LIN {X 0,Y 360.383,Z 396.223,A -85,B 0,C 180,E1 -13044.404,E2 -13044.404} C_VEL
LIN {X 0,Y 360.363,Z 398.205,A -85,B 0,C 180,E1 -13045.526,E2 -13045.526} C_VEL
LIN {X 0,Y 360.299,Z 399.765,A -85,B 0,C 180,E1 -13046.645,E2 -13046.645} C_VEL
LIN {X 0,Y 360.265,Z 400.875,A -85,B 0,C 180,E1 -13047.764,E2 -13047.764} C_VEL
LIN {X 0,Y 360.317,Z 401.567,A -85,B 0,C 180,E1 -13048.882,E2 -13048.882} C_VEL
LIN {X 0,Y 360.36,Z 401.867,A -85,B 0,C 180,E1 -13050,E2 -13050} C_VEL
LIN {X 0,Y 360.303,Z 401.773,A -85,B 0,C 180,E1 -13051.118,E2 -13051.118} C_VEL
LIN {X 0,Y 360.263,Z 401.25,A -85,B 0,C 180,E1 -13052.236,E2 -13052.236} C_VEL
LIN {X 0,Y 360.296,Z 400.314,A -85,B 0,C 180,E1 -13053.355,E2 -13053.355} C_VEL
LIN {X 0,Y 360.346,Z 398.979,A -85,B 0,C 180,E1 -13054.474,E2 -13054.474} C_VEL
LIN {X 0,Y 360.378,Z 396.542,A -85,B 0,C 180,E1 -13055.961,E2 -13055.961} C_VEL
LIN {X 0,Y 360.672,Z 392.315,A -85,B 0,C 180,E1 -13057.84,E2 -13057.84} C_VEL
LIN {X 0,Y 361.093,Z 387.341,A -85,B 0,C 180,E1 -13059.523,E2 -13059.523} C_VEL
LIN {X 0,Y 361.704,Z 381.091,A -85,B 0,C 180,E1 -13061.204,E2 -13061.204} C_VEL
LIN {X 0,Y 362.687,Z 373.329,A -85,B 0,C 180,E1 -13062.876,E2 -13062.876} C_VEL
LIN {X 0,Y 363.599,Z 365.4,A -85,B 0,C 180,E1 -13064.267,E2 -13064.267} C_VEL
LIN {X 0,Y 364.63,Z 355.745,A -85,B 0,C 180,E1 -13065.655,E2 -13065.655} C_VEL
LIN {X 0,Y 365.809,Z 345.051,A -85,B 0,C 180,E1 -13066.893,E2 -13066.893} C_VEL
LIN {X 0,Y 366.862,Z 334.733,A -85,B 0,C 180,E1 -13067.849,E2 -13067.849} C_VEL
LIN {X 0,Y 367.953,Z 323.553,A -85,B 0,C 180,E1 -13068.659,E2 -13068.659} C_VEL
LIN {X 0,Y 368.836,Z 310.34,A -85,B 0,C 180,E1 -13069.37,E2 -13069.37} C_VEL
LIN {X 0,Y 369.589,Z 297.288,A -85,B 0,C 180,E1 -13069.835,E2 -13069.835} C_VEL
LIN {X 0,Y 370.935,Z 222.024,A -85,B 0,C 180,E1 -13071.405,E2 -13071.405} C_VEL
LIN {X 0,Y 367.136,Z 199.174,A -85,B 0,C 180,E1 -13072.171,E2 -13072.171} C_VEL
LIN {X 0,Y 365.04,Z 188.802,A -85,B 0,C 180,E1 -13072.56,E2 -13072.56} C_VEL
LIN {X 0,Y 366.009,Z 179.574,A -85,B 0,C 180,E1 -13074.686,E2 -13074.686} C_VEL
LIN {X 0,Y 365.116,Z 173.255,A -85,B 0,C 180,E1 -13076.278,E2 -13076.278} C_VEL
LIN {X 0,Y 362.68,Z 161.895,A -85,B 0,C 180,E1 -13079.307,E2 -13079.307} C_VEL
LIN {X 0,Y 361.904,Z 158.409,A -85,B 0,C 180,E1 -13080.325,E2 -13080.325} C_VEL
LIN {X 0,Y 361.851,Z 158.414,A -85,B 0,C 180,E1 -13084.281,E2 -13084.281} C_VEL
LIN {X 0,Y 361.857,Z 158.413,A -85,B 0,C 180,E1 -13087.221,E2 -13087.221} C_VEL
LIN {X 0,Y 361.812,Z 158.419,A -85,B 0,C 180,E1 -13090.751,E2 -13090.751} C_VEL
LIN {X 0,Y 361.813,Z 158.416,A -85,B 0,C 180,E1 -13094.37,E2 -13094.37} C_VEL
LIN {X 0,Y 361.824,Z 158.414,A -85,B 0,C 180,E1 -13097.571,E2 -13097.571} C_VEL
LIN {X 0,Y 361.842,Z 158.412,A -85,B 0,C 180,E1 -13101.572,E2 -13101.572} C_VEL
LIN {X 0,Y 361.872,Z 158.408,A -85,B 0,C 180,E1 -13104.657,E2 -13104.657} C_VEL
LIN {X 0,Y 361.839,Z 158.41,A -85,B 0,C 180,E1 -13108.371,E2 -13108.371} C_VEL
LIN {X 0,Y 361.851,Z 158.404,A -85,B 0,C 180,E1 -13110.951,E2 -13110.951} C_VEL
LIN {X 0,Y 361.853,Z 158.403,A -85,B 0,C 180,E1 -13114.704,E2 -13114.704} C_VEL
LIN {X 0,Y 361.855,Z 158.408,A -85,B 0,C 180,E1 -13118.345,E2 -13118.345} C_VEL
LIN {X 0,Y 361.907,Z 158.405,A -85,B 0,C 180,E1 -13122.093,E2 -13122.093} C_VEL
LIN {X 0,Y 361.967,Z 158.398,A -85,B 0,C 180,E1 -13126.527,E2 -13126.527} C_VEL
LIN {X 0,Y 361.996,Z 158.385,A -85,B 0,C 180,E1 -13129.937,E2 -13129.937} C_VEL
LIN {X 0,Y 362.094,Z 158.377,A -85,B 0,C 180,E1 -13132.191,E2 -13132.191} C_VEL
LIN {X 0,Y 362.09,Z 158.375,A -85,B 0,C 180,E1 -13134.431,E2 -13134.431} C_VEL
LIN {X 0,Y 362.261,Z 158.351,A -85,B 0,C 180,E1 -13137.776,E2 -13137.776} C_VEL
LIN {X 0,Y 362.177,Z 158.365,A -85,B 0,C 180,E1 -13141.112,E2 -13141.112} C_VEL
LIN {X 0,Y 362.261,Z 158.354,A -85,B 0,C 180,E1 -13142.224,E2 -13142.224} C_VEL
LIN {X 0,Y 362.122,Z 158.376,A -85,B 0,C 180,E1 -13146.687,E2 -13146.687} C_VEL
LIN {X 0,Y 361.999,Z 158.391,A -85,B 0,C 180,E1 -13150.063,E2 -13150.063} C_VEL
LIN {X 0,Y 361.983,Z 158.397,A -85,B 0,C 180,E1 -13153.887,E2 -13153.887} C_VEL
LIN {X 0,Y 361.887,Z 158.405,A -85,B 0,C 180,E1 -13158.103,E2 -13158.103} C_VEL
LIN {X 0,Y 361.857,Z 158.414,A -85,B 0,C 180,E1 -13161.655,E2 -13161.655} C_VEL
LIN {X 0,Y 361.864,Z 158.414,A -85,B 0,C 180,E1 -13165.295,E2 -13165.295} C_VEL
LIN {X 0,Y 361.858,Z 158.412,A -85,B 0,C 180,E1 -13169.074,E2 -13169.074} C_VEL
LIN {X 0,Y 361.91,Z 158.531,A -85,B 0,C 180,E1 -13171.786,E2 -13171.786} C_VEL
LIN {X 0,Y 364.366,Z 169.922,A -85,B 0,C 180,E1 -13175.018,E2 -13175.018} C_VEL
LIN {X 0,Y 364.756,Z 171.823,A -85,B 0,C 180,E1 -13175.482,E2 -13175.482} C_VEL
LIN {X 0,Y 367.896,Z 180.526,A -85,B 0,C 180,E1 -13175.908,E2 -13175.908} C_VEL
LIN {X 0,Y 371.495,Z 197.463,A -85,B 0,C 180,E1 -13176.537,E2 -13176.537} C_VEL
LIN {X 0,Y 369.759,Z 279.168,A -85,B 0,C 180,E1 -13178.23,E2 -13178.23} C_VEL
LIN {X 0,Y 369.129,Z 292.46,A -85,B 0,C 180,E1 -13178.721,E2 -13178.721} C_VEL
LIN {X 0,Y 368.436,Z 305.031,A -85,B 0,C 180,E1 -13179.416,E2 -13179.416} C_VEL
LIN {X 0,Y 367.469,Z 316.572,A -85,B 0,C 180,E1 -13180.272,E2 -13180.272} C_VEL
LIN {X 0,Y 366.343,Z 328.059,A -85,B 0,C 180,E1 -13181.373,E2 -13181.373} C_VEL
LIN {X 0,Y 365.194,Z 338.479,A -85,B 0,C 180,E1 -13182.626,E2 -13182.626} C_VEL
LIN {X 0,Y 364.038,Z 348.321,A -85,B 0,C 180,E1 -13184.112,E2 -13184.112} C_VEL
LIN {X 0,Y 362.998,Z 357.318,A -85,B 0,C 180,E1 -13185.813,E2 -13185.813} C_VEL
LIN {X 0,Y 362.078,Z 364.557,A -85,B 0,C 180,E1 -13187.527,E2 -13187.527} C_VEL
LIN {X 0,Y 361.392,Z 370.511,A -85,B 0,C 180,E1 -13189.327,E2 -13189.327} C_VEL
LIN {X 0,Y 360.886,Z 375.198,A -85,B 0,C 180,E1 -13191.167,E2 -13191.167} C_VEL
LIN {X 0,Y 360.496,Z 378.709,A -85,B 0,C 180,E1 -13193.065,E2 -13193.065} C_VEL
LIN {X 0,Y 360.179,Z 381.055,A -85,B 0,C 180,E1 -13195.038,E2 -13195.038} C_VEL
LIN {X 0,Y 360.074,Z 382.107,A -85,B 0,C 180,E1 -13197.065,E2 -13197.065} C_VEL
LIN {X 0,Y 360.104,Z 381.816,A -85,B 0,C 180,E1 -13199.175,E2 -13199.175} C_VEL
LIN {X 0,Y 360.268,Z 380.007,A -85,B 0,C 180,E1 -13201.384,E2 -13201.384} C_VEL
LIN {X 0,Y 360.569,Z 376.96,A -85,B 0,C 180,E1 -13203.365,E2 -13203.365} C_VEL
LIN {X 0,Y 360.916,Z 372.764,A -85,B 0,C 180,E1 -13205.25,E2 -13205.25} C_VEL
LIN {X 0,Y 361.336,Z 367.249,A -85,B 0,C 180,E1 -13207.107,E2 -13207.107} C_VEL
LIN {X 0,Y 361.938,Z 360.996,A -85,B 0,C 180,E1 -13208.757,E2 -13208.757} C_VEL
LIN {X 0,Y 362.777,Z 352.79,A -85,B 0,C 180,E1 -13210.477,E2 -13210.477} C_VEL
LIN {X 0,Y 363.701,Z 343.833,A -85,B 0,C 180,E1 -13211.99,E2 -13211.99} C_VEL
LIN {X 0,Y 364.645,Z 334.126,A -85,B 0,C 180,E1 -13213.321,E2 -13213.321} C_VEL
LIN {X 0,Y 365.693,Z 322.992,A -85,B 0,C 180,E1 -13214.535,E2 -13214.535} C_VEL
LIN {X 0,Y 366.566,Z 311.016,A -85,B 0,C 180,E1 -13215.567,E2 -13215.567} C_VEL
LIN {X 0,Y 367.308,Z 298.616,A -85,B 0,C 180,E1 -13216.374,E2 -13216.374} C_VEL
LIN {X 0,Y 368.004,Z 285.25,A -85,B 0,C 180,E1 -13216.981,E2 -13216.981} C_VEL
LIN {X 0,Y 368.435,Z 272.362,A -85,B 0,C 180,E1 -13217.347,E2 -13217.347} C_VEL
LIN {X 0,Y 369.683,Z 196.406,A -85,B 0,C 180,E1 -13218.884,E2 -13218.884} C_VEL
LIN {X 0,Y 364.942,Z 172.85,A -85,B 0,C 180,E1 -13219.651,E2 -13219.651} C_VEL
LIN {X 0,Y 364.418,Z 171.078,A -85,B 0,C 180,E1 -13219.724,E2 -13219.724} C_VEL
LIN {X 0,Y 362.13,Z 158.379,A -85,B 0,C 180,E1 -13223.243,E2 -13223.243} C_VEL
LIN {X 0,Y 362.279,Z 158.355,A -85,B 0,C 180,E1 -13227.776,E2 -13227.776} C_VEL
LIN {X 0,Y 362.206,Z 158.364,A -85,B 0,C 180,E1 -13231.112,E2 -13231.112} C_VEL
LIN {X 0,Y 362.267,Z 158.361,A -85,B 0,C 180,E1 -13232.224,E2 -13232.224} C_VEL
LIN {X 0,Y 362.124,Z 158.376,A -85,B 0,C 180,E1 -13236.687,E2 -13236.687} C_VEL
LIN {X 0,Y 362.03,Z 158.391,A -85,B 0,C 180,E1 -13240.062,E2 -13240.062} C_VEL
LIN {X 0,Y 361.973,Z 158.392,A -85,B 0,C 180,E1 -13240.987,E2 -13240.987} C_VEL
LIN {X 0,Y 361.296,Z 158.481,A -85,B 0,C 180,E1 -13241.916,E2 -13241.916} C_VEL
LIN {X 0,Y 358.408,Z 158.838,A -85,B 0,C 180,E1 -13243.426,E2 -13243.426} C_VEL
LIN {X 0,Y 355.968,Z 159.142,A -85,B 0,C 180,E1 -13244.648,E2 -13244.648} C_VEL
LIN {X 0,Y 354.927,Z 159.273,A -85,B 0,C 180,E1 -13245.594,E2 -13245.594} C_VEL
LIN {X 0,Y 354.847,Z 159.283,A -85,B 0,C 180,E1 -13245.914,E2 -13245.914} C_VEL
LIN {X 0,Y 354.849,Z 159.281,A -85,B 0,C 180,E1 -13248.475,E2 -13248.475} C_VEL
LIN {X 0,Y 354.809,Z 159.288,A -85,B 0,C 180,E1 -13252.108,E2 -13252.108} C_VEL
LIN {X 0,Y 354.805,Z 159.291,A -85,B 0,C 180,E1 -13255.835,E2 -13255.835} C_VEL
LIN {X 0,Y 354.798,Z 159.292,A -85,B 0,C 180,E1 -13259.684,E2 -13259.684} C_VEL
LIN {X 0,Y 354.789,Z 159.288,A -85,B 0,C 180,E1 -13262.334,E2 -13262.334} C_VEL
LIN {X 0,Y 354.823,Z 159.287,A -85,B 0,C 180,E1 -13265.699,E2 -13265.699} C_VEL
LIN {X 0,Y 354.77,Z 159.296,A -85,B 0,C 180,E1 -13269.413,E2 -13269.413} C_VEL
LIN {X 0,Y 354.787,Z 159.29,A -85,B 0,C 180,E1 -13272.867,E2 -13272.867} C_VEL
LIN {X 0,Y 354.765,Z 159.291,A -85,B 0,C 180,E1 -13276.103,E2 -13276.103} C_VEL
LIN {X 0,Y 354.768,Z 159.296,A -85,B 0,C 180,E1 -13279.176,E2 -13279.176} C_VEL
LIN {X 0,Y 354.802,Z 159.286,A -85,B 0,C 180,E1 -13282.404,E2 -13282.404} C_VEL
LIN {X 0,Y 354.811,Z 159.29,A -85,B 0,C 180,E1 -13284.94,E2 -13284.94} C_VEL
LIN {X 0,Y 354.796,Z 159.288,A -85,B 0,C 180,E1 -13288.405,E2 -13288.405} C_VEL
LIN {X 0,Y 354.802,Z 159.286,A -85,B 0,C 180,E1 -13291.615,E2 -13291.615} C_VEL
LIN {X 0,Y 354.837,Z 159.282,A -85,B 0,C 180,E1 -13295.657,E2 -13295.657} C_VEL
LIN {X 0,Y 354.827,Z 159.285,A -85,B 0,C 180,E1 -13299.113,E2 -13299.113} C_VEL
LIN {X 0,Y 354.855,Z 159.284,A -85,B 0,C 180,E1 -13302.718,E2 -13302.718} C_VEL
LIN {X 0,Y 354.943,Z 159.272,A -85,B 0,C 180,E1 -13306.255,E2 -13306.255} C_VEL
LIN {X 0,Y 354.958,Z 159.267,A -85,B 0,C 180,E1 -13309.735,E2 -13309.735} C_VEL
LIN {X 0,Y 355.091,Z 159.25,A -85,B 0,C 180,E1 -13313.18,E2 -13313.18} C_VEL
LIN {X 0,Y 355.23,Z 159.234,A -85,B 0,C 180,E1 -13317.732,E2 -13317.732} C_VEL
LIN {X 0,Y 355.149,Z 159.243,A -85,B 0,C 180,E1 -13321.134,E2 -13321.134} C_VEL
LIN {X 0,Y 355.229,Z 159.238,A -85,B 0,C 180,E1 -13322.268,E2 -13322.268} C_VEL
LIN {X 0,Y 355.091,Z 159.25,A -85,B 0,C 180,E1 -13326.82,E2 -13326.82} C_VEL
LIN {X 0,Y 354.953,Z 159.27,A -85,B 0,C 180,E1 -13330.265,E2 -13330.265} C_VEL
LIN {X 0,Y 354.895,Z 159.279,A -85,B 0,C 180,E1 -13333.986,E2 -13333.986} C_VEL
LIN {X 0,Y 354.837,Z 159.285,A -85,B 0,C 180,E1 -13338.064,E2 -13338.064} C_VEL
LIN {X 0,Y 354.808,Z 159.287,A -85,B 0,C 180,E1 -13342.108,E2 -13342.108} C_VEL
LIN {X 0,Y 354.797,Z 159.29,A -85,B 0,C 180,E1 -13345.835,E2 -13345.835} C_VEL
LIN {X 0,Y 354.795,Z 159.291,A -85,B 0,C 180,E1 -13349.684,E2 -13349.684} C_VEL
LIN {X 0,Y 354.788,Z 159.288,A -85,B 0,C 180,E1 -13352.333,E2 -13352.333} C_VEL
LIN {X 0,Y 354.82,Z 159.286,A -85,B 0,C 180,E1 -13355.698,E2 -13355.698} C_VEL
LIN {X 0,Y 354.77,Z 159.294,A -85,B 0,C 180,E1 -13359.412,E2 -13359.412} C_VEL
LIN {X 0,Y 354.783,Z 159.292,A -85,B 0,C 180,E1 -13362.866,E2 -13362.866} C_VEL
LIN {X 0,Y 354.764,Z 159.291,A -85,B 0,C 180,E1 -13366.103,E2 -13366.103} C_VEL
LIN {X 0,Y 354.764,Z 159.295,A -85,B 0,C 180,E1 -13369.175,E2 -13369.175} C_VEL
LIN {X 0,Y 354.8,Z 159.288,A -85,B 0,C 180,E1 -13372.404,E2 -13372.404} C_VEL
LIN {X 0,Y 354.809,Z 159.29,A -85,B 0,C 180,E1 -13374.94,E2 -13374.94} C_VEL
LIN {X 0,Y 354.777,Z 159.292,A -85,B 0,C 180,E1 -13378.41,E2 -13378.41} C_VEL
LIN {X 0,Y 354.854,Z 159.395,A -85,B 0,C 180,E1 -13380.321,E2 -13380.321} C_VEL
LIN {X 0,Y 357.448,Z 172.358,A -85,B 0,C 180,E1 -13383.744,E2 -13383.744} C_VEL
LIN {X 0,Y 358.451,Z 178.801,A -85,B 0,C 180,E1 -13385.377,E2 -13385.377} C_VEL
LIN {X 0,Y 357.438,Z 189.546,A -85,B 0,C 180,E1 -13387.906,E2 -13387.906} C_VEL
LIN {X 0,Y 362.684,Z 223.59,A -85,B 0,C 180,E1 -13388.946,E2 -13388.946} C_VEL
LIN {X 0,Y 361.286,Z 298.073,A -85,B 0,C 180,E1 -13390.504,E2 -13390.504} C_VEL
LIN {X 0,Y 360.646,Z 311.829,A -85,B 0,C 180,E1 -13391.023,E2 -13391.023} C_VEL
LIN {X 0,Y 359.793,Z 324.254,A -85,B 0,C 180,E1 -13391.714,E2 -13391.714} C_VEL
LIN {X 0,Y 358.739,Z 336.164,A -85,B 0,C 180,E1 -13392.617,E2 -13392.617} C_VEL
LIN {X 0,Y 357.646,Z 347.626,A -85,B 0,C 180,E1 -13393.738,E2 -13393.738} C_VEL
LIN {X 0,Y 356.733,Z 357.74,A -85,B 0,C 180,E1 -13394.981,E2 -13394.981} C_VEL
LIN {X 0,Y 355.837,Z 366.43,A -85,B 0,C 180,E1 -13396.29,E2 -13396.29} C_VEL
LIN {X 0,Y 354.87,Z 375.592,A -85,B 0,C 180,E1 -13397.998,E2 -13397.998} C_VEL
LIN {X 0,Y 354.199,Z 382.972,A -85,B 0,C 180,E1 -13399.713,E2 -13399.713} C_VEL
LIN {X 0,Y 353.712,Z 388.878,A -85,B 0,C 180,E1 -13401.43,E2 -13401.43} C_VEL
LIN {X 0,Y 353.415,Z 393.517,A -85,B 0,C 180,E1 -13403.147,E2 -13403.147} C_VEL
LIN {X 0,Y 353.29,Z 395.958,A -85,B 0,C 180,E1 -13404.292,E2 -13404.292} C_VEL
LIN {X 0,Y 353.276,Z 397.953,A -85,B 0,C 180,E1 -13405.436,E2 -13405.436} C_VEL
LIN {X 0,Y 353.221,Z 399.525,A -85,B 0,C 180,E1 -13406.578,E2 -13406.578} C_VEL
LIN {X 0,Y 353.173,Z 400.655,A -85,B 0,C 180,E1 -13407.719,E2 -13407.719} C_VEL
LIN {X 0,Y 353.217,Z 401.357,A -85,B 0,C 180,E1 -13408.86,E2 -13408.86} C_VEL
LIN {X 0,Y 353.263,Z 401.667,A -85,B 0,C 180,E1 -13410,E2 -13410} C_VEL
LIN {X 0,Y 353.203,Z 401.582,A -85,B 0,C 180,E1 -13411.14,E2 -13411.14} C_VEL
LIN {X 0,Y 353.171,Z 401.078,A -85,B 0,C 180,E1 -13412.281,E2 -13412.281} C_VEL
LIN {X 0,Y 353.217,Z 400.15,A -85,B 0,C 180,E1 -13413.422,E2 -13413.422} C_VEL
LIN {X 0,Y 353.259,Z 398.824,A -85,B 0,C 180,E1 -13414.564,E2 -13414.564} C_VEL
LIN {X 0,Y 353.275,Z 396.743,A -85,B 0,C 180,E1 -13415.904,E2 -13415.904} C_VEL
LIN {X 0,Y 353.617,Z 392.206,A -85,B 0,C 180,E1 -13417.997,E2 -13417.997} C_VEL
LIN {X 0,Y 354.057,Z 387.261,A -85,B 0,C 180,E1 -13419.714,E2 -13419.714} C_VEL
LIN {X 0,Y 354.705,Z 381.047,A -85,B 0,C 180,E1 -13421.428,E2 -13421.428} C_VEL
LIN {X 0,Y 355.758,Z 373.33,A -85,B 0,C 180,E1 -13423.131,E2 -13423.131} C_VEL
LIN {X 0,Y 356.691,Z 365.443,A -85,B 0,C 180,E1 -13424.55,E2 -13424.55} C_VEL
LIN {X 0,Y 357.788,Z 355.834,A -85,B 0,C 180,E1 -13425.962,E2 -13425.962} C_VEL
LIN {X 0,Y 359.022,Z 345.198,A -85,B 0,C 180,E1 -13427.222,E2 -13427.222} C_VEL
LIN {X 0,Y 360.301,Z 333.295,A -85,B 0,C 180,E1 -13428.333,E2 -13428.333} C_VEL
LIN {X 0,Y 361.462,Z 321.711,A -85,B 0,C 180,E1 -13429.154,E2 -13429.154} C_VEL
LIN {X 0,Y 362.293,Z 309.448,A -85,B 0,C 180,E1 -13429.808,E2 -13429.808} C_VEL
LIN {X 0,Y 363.033,Z 295.927,A -85,B 0,C 180,E1 -13430.283,E2 -13430.283} C_VEL
LIN {X 0,Y 364.513,Z 223.491,A -85,B 0,C 180,E1 -13431.811,E2 -13431.811} C_VEL
LIN {X 0,Y 360.759,Z 200.666,A -85,B 0,C 180,E1 -13432.6,E2 -13432.6} C_VEL
LIN {X 0,Y 358.309,Z 188.45,A -85,B 0,C 180,E1 -13433.097,E2 -13433.097} C_VEL
LIN {X 0,Y 359.142,Z 180.87,A -85,B 0,C 180,E1 -13434.881,E2 -13434.881} C_VEL
LIN {X 0,Y 357.922,Z 173.312,A -85,B 0,C 180,E1 -13436.848,E2 -13436.848} C_VEL
LIN {X 0,Y 355.184,Z 160.771,A -85,B 0,C 180,E1 -13440.302,E2 -13440.302} C_VEL
LIN {X 0,Y 354.843,Z 159.288,A -85,B 0,C 180,E1 -13440.747,E2 -13440.747} C_VEL
LIN {X 0,Y 354.808,Z 159.293,A -85,B 0,C 180,E1 -13443.702,E2 -13443.702} C_VEL
LIN {X 0,Y 354.792,Z 159.289,A -85,B 0,C 180,E1 -13446.461,E2 -13446.461} C_VEL
LIN {X 0,Y 354.77,Z 159.295,A -85,B 0,C 180,E1 -13449.413,E2 -13449.413} C_VEL
LIN {X 0,Y 354.783,Z 159.295,A -85,B 0,C 180,E1 -13452.866,E2 -13452.866} C_VEL
LIN {X 0,Y 354.764,Z 159.295,A -85,B 0,C 180,E1 -13456.103,E2 -13456.103} C_VEL
LIN {X 0,Y 354.765,Z 159.292,A -85,B 0,C 180,E1 -13459.176,E2 -13459.176} C_VEL
LIN {X 0,Y 354.8,Z 159.29,A -85,B 0,C 180,E1 -13462.405,E2 -13462.405} C_VEL
LIN {X 0,Y 354.81,Z 159.291,A -85,B 0,C 180,E1 -13464.94,E2 -13464.94} C_VEL
LIN {X 0,Y 354.795,Z 159.288,A -85,B 0,C 180,E1 -13468.406,E2 -13468.406} C_VEL
LIN {X 0,Y 354.791,Z 159.284,A -85,B 0,C 180,E1 -13471.614,E2 -13471.614} C_VEL
LIN {X 0,Y 354.804,Z 159.28,A -85,B 0,C 180,E1 -13475.419,E2 -13475.419} C_VEL
LIN {X 0,Y 354.82,Z 159.276,A -85,B 0,C 180,E1 -13479.113,E2 -13479.113} C_VEL
LIN {X 0,Y 354.845,Z 159.281,A -85,B 0,C 180,E1 -13482.717,E2 -13482.717} C_VEL
LIN {X 0,Y 354.911,Z 159.275,A -85,B 0,C 180,E1 -13486.254,E2 -13486.254} C_VEL
LIN {X 0,Y 354.952,Z 159.261,A -85,B 0,C 180,E1 -13489.735,E2 -13489.735} C_VEL
LIN {X 0,Y 355.091,Z 159.241,A -85,B 0,C 180,E1 -13493.18,E2 -13493.18} C_VEL
LIN {X 0,Y 355.223,Z 159.227,A -85,B 0,C 180,E1 -13497.732,E2 -13497.732} C_VEL
LIN {X 0,Y 355.149,Z 159.24,A -85,B 0,C 180,E1 -13501.134,E2 -13501.134} C_VEL
LIN {X 0,Y 355.223,Z 159.23,A -85,B 0,C 180,E1 -13502.268,E2 -13502.268} C_VEL
LIN {X 0,Y 355.089,Z 159.252,A -85,B 0,C 180,E1 -13506.82,E2 -13506.82} C_VEL
LIN {X 0,Y 354.955,Z 159.27,A -85,B 0,C 180,E1 -13510.265,E2 -13510.265} C_VEL
LIN {X 0,Y 354.927,Z 159.277,A -85,B 0,C 180,E1 -13514.006,E2 -13514.006} C_VEL
LIN {X 0,Y 354.845,Z 159.282,A -85,B 0,C 180,E1 -13518.068,E2 -13518.068} C_VEL
LIN {X 0,Y 354.81,Z 159.288,A -85,B 0,C 180,E1 -13522.108,E2 -13522.108} C_VEL
LIN {X 0,Y 354.803,Z 159.293,A -85,B 0,C 180,E1 -13525.835,E2 -13525.835} C_VEL
LIN {X 0,Y 354.799,Z 159.292,A -85,B 0,C 180,E1 -13529.684,E2 -13529.684} C_VEL
LIN {X 0,Y 354.861,Z 159.332,A -85,B 0,C 180,E1 -13531.312,E2 -13531.312} C_VEL
LIN {X 0,Y 357.081,Z 169.36,A -85,B 0,C 180,E1 -13534.244,E2 -13534.244} C_VEL
LIN {X 0,Y 357.543,Z 171.759,A -85,B 0,C 180,E1 -13534.924,E2 -13534.924} C_VEL
LIN {X 0,Y 361.629,Z 182.544,A -85,B 0,C 180,E1 -13535.493,E2 -13535.493} C_VEL
LIN {X 0,Y 365.078,Z 199.281,A -85,B 0,C 180,E1 -13536.126,E2 -13536.126} C_VEL
LIN {X 0,Y 363.191,Z 279.325,A -85,B 0,C 180,E1 -13537.815,E2 -13537.815} C_VEL
LIN {X 0,Y 362.495,Z 293.318,A -85,B 0,C 180,E1 -13538.346,E2 -13538.346} C_VEL
LIN {X 0,Y 361.731,Z 306.162,A -85,B 0,C 180,E1 -13539.085,E2 -13539.085} C_VEL
LIN {X 0,Y 360.654,Z 318.22,A -85,B 0,C 180,E1 -13540.021,E2 -13540.021} C_VEL
LIN {X 0,Y 359.486,Z 329.482,A -85,B 0,C 180,E1 -13541.146,E2 -13541.146} C_VEL
LIN {X 0,Y 358.277,Z 339.732,A -85,B 0,C 180,E1 -13542.433,E2 -13542.433} C_VEL
LIN {X 0,Y 357.226,Z 348.373,A -85,B 0,C 180,E1 -13543.774,E2 -13543.774} C_VEL
LIN {X 0,Y 356.096,Z 357.557,A -85,B 0,C 180,E1 -13545.54,E2 -13545.54} C_VEL
LIN {X 0,Y 355.068,Z 365.081,A -85,B 0,C 180,E1 -13547.369,E2 -13547.369} C_VEL
LIN {X 0,Y 354.372,Z 370.735,A -85,B 0,C 180,E1 -13549.12,E2 -13549.12} C_VEL
LIN {X 0,Y 353.915,Z 374.891,A -85,B 0,C 180,E1 -13550.756,E2 -13550.756} C_VEL
LIN {X 0,Y 353.497,Z 378.522,A -85,B 0,C 180,E1 -13552.68,E2 -13552.68} C_VEL
LIN {X 0,Y 353.138,Z 381.069,A -85,B 0,C 180,E1 -13554.75,E2 -13554.75} C_VEL
LIN {X 0,Y 352.974,Z 382.256,A -85,B 0,C 180,E1 -13556.747,E2 -13556.747} C_VEL
LIN {X 0,Y 353.002,Z 382.134,A -85,B 0,C 180,E1 -13558.882,E2 -13558.882} C_VEL
LIN {X 0,Y 353.144,Z 380.514,A -85,B 0,C 180,E1 -13561.123,E2 -13561.123} C_VEL
LIN {X 0,Y 353.488,Z 377.091,A -85,B 0,C 180,E1 -13563.468,E2 -13563.468} C_VEL
LIN {X 0,Y 353.847,Z 372.977,A -85,B 0,C 180,E1 -13565.348,E2 -13565.348} C_VEL
LIN {X 0,Y 354.292,Z 367.466,A -85,B 0,C 180,E1 -13567.243,E2 -13567.243} C_VEL
LIN {X 0,Y 355.029,Z 360.353,A -85,B 0,C 180,E1 -13569.125,E2 -13569.125} C_VEL
LIN {X 0,Y 355.946,Z 351.924,A -85,B 0,C 180,E1 -13570.885,E2 -13570.885} C_VEL
LIN {X 0,Y 356.995,Z 342.024,A -85,B 0,C 180,E1 -13572.529,E2 -13572.529} C_VEL
LIN {X 0,Y 358.004,Z 331.652,A -85,B 0,C 180,E1 -13573.901,E2 -13573.901} C_VEL
LIN {X 0,Y 359.048,Z 320.166,A -85,B 0,C 180,E1 -13575.113,E2 -13575.113} C_VEL
LIN {X 0,Y 359.981,Z 308.137,A -85,B 0,C 180,E1 -13576.091,E2 -13576.091} C_VEL
LIN {X 0,Y 360.655,Z 296.27,A -85,B 0,C 180,E1 -13576.825,E2 -13576.825} C_VEL
LIN {X 0,Y 361.311,Z 283.385,A -85,B 0,C 180,E1 -13577.385,E2 -13577.385} C_VEL
LIN {X 0,Y 361.7,Z 268.315,A -85,B 0,C 180,E1 -13577.77,E2 -13577.77} C_VEL
LIN {X 0,Y 363.009,Z 197.553,A -85,B 0,C 180,E1 -13579.225,E2 -13579.225} C_VEL
LIN {X 0,Y 358.504,Z 175.134,A -85,B 0,C 180,E1 -13579.971,E2 -13579.971} C_VEL
LIN {X 0,Y 357.234,Z 171.176,A -85,B 0,C 180,E1 -13580.159,E2 -13580.159} C_VEL
LIN {X 0,Y 355.077,Z 159.258,A -85,B 0,C 180,E1 -13583.536,E2 -13583.536} C_VEL
LIN {X 0,Y 355.242,Z 159.232,A -85,B 0,C 180,E1 -13587.732,E2 -13587.732} C_VEL
LIN {X 0,Y 355.174,Z 159.24,A -85,B 0,C 180,E1 -13591.134,E2 -13591.134} C_VEL
LIN {X 0,Y 355.23,Z 159.238,A -85,B 0,C 180,E1 -13592.268,E2 -13592.268} C_VEL
LIN {X 0,Y 355.09,Z 159.251,A -85,B 0,C 180,E1 -13596.82,E2 -13596.82} C_VEL
LIN {X 0,Y 354.978,Z 159.269,A -85,B 0,C 180,E1 -13600.264,E2 -13600.264} C_VEL
LIN {X 0,Y 354.926,Z 159.276,A -85,B 0,C 180,E1 -13604.006,E2 -13604.006} C_VEL
LIN {X 0,Y 354.847,Z 159.283,A -85,B 0,C 180,E1 -13605.914,E2 -13605.914} C_VEL
LIN {X 0,Y 354.185,Z 159.372,A -85,B 0,C 180,E1 -13606.862,E2 -13606.862} C_VEL
LIN {X 0,Y 351.315,Z 159.729,A -85,B 0,C 180,E1 -13608.402,E2 -13608.402} C_VEL
LIN {X 0,Y 348.885,Z 160.027,A -85,B 0,C 180,E1 -13609.648,E2 -13609.648} C_VEL
LIN {X 0,Y 347.85,Z 160.153,A -85,B 0,C 180,E1 -13610.613,E2 -13610.613} C_VEL
LIN {X 0,Y 347.77,Z 160.162,A -85,B 0,C 180,E1 -13610.94,E2 -13610.94} C_VEL
LIN {X 0,Y 347.773,Z 160.162,A -85,B 0,C 180,E1 -13614.579,E2 -13614.579} C_VEL
LIN {X 0,Y 347.738,Z 160.172,A -85,B 0,C 180,E1 -13617.7,E2 -13617.7} C_VEL
LIN {X 0,Y 347.74,Z 160.166,A -85,B 0,C 180,E1 -13620.349,E2 -13620.349} C_VEL
LIN {X 0,Y 347.751,Z 160.166,A -85,B 0,C 180,E1 -13624.044,E2 -13624.044} C_VEL
LIN {X 0,Y 347.758,Z 160.168,A -85,B 0,C 180,E1 -13627.322,E2 -13627.322} C_VEL
LIN {X 0,Y 347.743,Z 160.169,A -85,B 0,C 180,E1 -13631.601,E2 -13631.601} C_VEL
LIN {X 0,Y 347.705,Z 160.174,A -85,B 0,C 180,E1 -13635.027,E2 -13635.027} C_VEL
LIN {X 0,Y 347.743,Z 160.166,A -85,B 0,C 180,E1 -13638.399,E2 -13638.399} C_VEL
LIN {X 0,Y 347.758,Z 160.166,A -85,B 0,C 180,E1 -13642.679,E2 -13642.679} C_VEL
LIN {X 0,Y 347.751,Z 160.164,A -85,B 0,C 180,E1 -13645.956,E2 -13645.956} C_VEL
LIN {X 0,Y 347.741,Z 160.166,A -85,B 0,C 180,E1 -13649.651,E2 -13649.651} C_VEL
LIN {X 0,Y 347.751,Z 160.165,A -85,B 0,C 180,E1 -13653.601,E2 -13653.601} C_VEL
LIN {X 0,Y 347.766,Z 160.163,A -85,B 0,C 180,E1 -13656.16,E2 -13656.16} C_VEL
LIN {X 0,Y 347.78,Z 160.161,A -85,B 0,C 180,E1 -13659.907,E2 -13659.907} C_VEL
LIN {X 0,Y 347.8,Z 160.158,A -85,B 0,C 180,E1 -13663.567,E2 -13663.567} C_VEL
LIN {X 0,Y 347.891,Z 160.148,A -85,B 0,C 180,E1 -13667.16,E2 -13667.16} C_VEL
LIN {X 0,Y 347.938,Z 160.144,A -85,B 0,C 180,E1 -13670.701,E2 -13670.701} C_VEL
LIN {X 0,Y 348.043,Z 160.133,A -85,B 0,C 180,E1 -13674.205,E2 -13674.205} C_VEL
LIN {X 0,Y 348.191,Z 160.111,A -85,B 0,C 180,E1 -13677.686,E2 -13677.686} C_VEL
LIN {X 0,Y 348.12,Z 160.118,A -85,B 0,C 180,E1 -13681.157,E2 -13681.157} C_VEL
LIN {X 0,Y 348.19,Z 160.114,A -85,B 0,C 180,E1 -13682.314,E2 -13682.314} C_VEL
LIN {X 0,Y 348.062,Z 160.126,A -85,B 0,C 180,E1 -13686.959,E2 -13686.959} C_VEL
LIN {X 0,Y 347.892,Z 160.148,A -85,B 0,C 180,E1 -13690.475,E2 -13690.475} C_VEL
LIN {X 0,Y 347.854,Z 160.155,A -85,B 0,C 180,E1 -13694.119,E2 -13694.119} C_VEL
LIN {X 0,Y 347.79,Z 160.161,A -85,B 0,C 180,E1 -13698.238,E2 -13698.238} C_VEL
LIN {X 0,Y 347.766,Z 160.168,A -85,B 0,C 180,E1 -13701.624,E2 -13701.624} C_VEL
LIN {X 0,Y 347.736,Z 160.168,A -85,B 0,C 180,E1 -13705.114,E2 -13705.114} C_VEL
LIN {X 0,Y 347.727,Z 160.171,A -85,B 0,C 180,E1 -13707.701,E2 -13707.701} C_VEL
LIN {X 0,Y 347.738,Z 160.166,A -85,B 0,C 180,E1 -13710.349,E2 -13710.349} C_VEL
LIN {X 0,Y 347.75,Z 160.165,A -85,B 0,C 180,E1 -13714.043,E2 -13714.043} C_VEL
LIN {X 0,Y 347.756,Z 160.169,A -85,B 0,C 180,E1 -13717.322,E2 -13717.322} C_VEL
LIN {X 0,Y 347.697,Z 160.171,A -85,B 0,C 180,E1 -13720.302,E2 -13720.302} C_VEL
LIN {X 0,Y 347.722,Z 160.171,A -85,B 0,C 180,E1 -13723.408,E2 -13723.408} C_VEL
LIN {X 0,Y 347.724,Z 160.17,A -85,B 0,C 180,E1 -13726.687,E2 -13726.687} C_VEL
LIN {X 0,Y 347.702,Z 160.171,A -85,B 0,C 180,E1 -13730.182,E2 -13730.182} C_VEL
LIN {X 0,Y 347.755,Z 160.167,A -85,B 0,C 180,E1 -13732.678,E2 -13732.678} C_VEL
LIN {X 0,Y 347.749,Z 160.165,A -85,B 0,C 180,E1 -13735.956,E2 -13735.956} C_VEL
LIN {X 0,Y 347.819,Z 160.26,A -85,B 0,C 180,E1 -13739.998,E2 -13739.998} C_VEL
LIN {X 0,Y 350.394,Z 173.226,A -85,B 0,C 180,E1 -13743.495,E2 -13743.495} C_VEL
LIN {X 0,Y 351.497,Z 179.678,A -85,B 0,C 180,E1 -13745.172,E2 -13745.172} C_VEL
LIN {X 0,Y 350.589,Z 189.358,A -85,B 0,C 180,E1 -13747.498,E2 -13747.498} C_VEL
LIN {X 0,Y 355.895,Z 223.535,A -85,B 0,C 180,E1 -13748.575,E2 -13748.575} C_VEL
LIN {X 0,Y 354.526,Z 297.499,A -85,B 0,C 180,E1 -13750.155,E2 -13750.155} C_VEL
LIN {X 0,Y 353.922,Z 310.623,A -85,B 0,C 180,E1 -13750.648,E2 -13750.648} C_VEL
LIN {X 0,Y 353.047,Z 323.321,A -85,B 0,C 180,E1 -13751.352,E2 -13751.352} C_VEL
LIN {X 0,Y 351.955,Z 335.446,A -85,B 0,C 180,E1 -13752.271,E2 -13752.271} C_VEL
LIN {X 0,Y 350.827,Z 347.009,A -85,B 0,C 180,E1 -13753.413,E2 -13753.413} C_VEL
LIN {X 0,Y 349.873,Z 356.775,A -85,B 0,C 180,E1 -13754.621,E2 -13754.621} C_VEL
LIN {X 0,Y 348.897,Z 365.966,A -85,B 0,C 180,E1 -13756.012,E2 -13756.012} C_VEL
LIN {X 0,Y 348.057,Z 373.819,A -85,B 0,C 180,E1 -13757.463,E2 -13757.463} C_VEL
LIN {X 0,Y 347.256,Z 381.479,A -85,B 0,C 180,E1 -13759.21,E2 -13759.21} C_VEL
LIN {X 0,Y 346.666,Z 388.552,A -85,B 0,C 180,E1 -13761.254,E2 -13761.254} C_VEL
LIN {X 0,Y 346.341,Z 393.224,A -85,B 0,C 180,E1 -13763.007,E2 -13763.007} C_VEL
LIN {X 0,Y 346.176,Z 396.346,A -85,B 0,C 180,E1 -13764.531,E2 -13764.531} C_VEL
LIN {X 0,Y 346.145,Z 399.28,A -85,B 0,C 180,E1 -13766.508,E2 -13766.508} C_VEL
LIN {X 0,Y 346.085,Z 400.433,A -85,B 0,C 180,E1 -13767.672,E2 -13767.672} C_VEL
LIN {X 0,Y 346.117,Z 401.145,A -85,B 0,C 180,E1 -13768.837,E2 -13768.837} C_VEL
LIN {X 0,Y 346.165,Z 401.465,A -85,B 0,C 180,E1 -13770,E2 -13770} C_VEL
LIN {X 0,Y 346.103,Z 401.391,A -85,B 0,C 180,E1 -13771.164,E2 -13771.164} C_VEL
LIN {X 0,Y 346.082,Z 400.909,A -85,B 0,C 180,E1 -13772.328,E2 -13772.328} C_VEL
LIN {X 0,Y 346.141,Z 399.994,A -85,B 0,C 180,E1 -13773.492,E2 -13773.492} C_VEL
LIN {X 0,Y 346.157,Z 398.679,A -85,B 0,C 180,E1 -13774.658,E2 -13774.658} C_VEL
LIN {X 0,Y 346.241,Z 395.908,A -85,B 0,C 180,E1 -13776.409,E2 -13776.409} C_VEL
LIN {X 0,Y 346.562,Z 392.11,A -85,B 0,C 180,E1 -13778.161,E2 -13778.161} C_VEL
LIN {X 0,Y 347.038,Z 387.19,A -85,B 0,C 180,E1 -13779.912,E2 -13779.912} C_VEL
LIN {X 0,Y 347.717,Z 381.003,A -85,B 0,C 180,E1 -13781.661,E2 -13781.661} C_VEL
LIN {X 0,Y 348.811,Z 373.326,A -85,B 0,C 180,E1 -13783.398,E2 -13783.398} C_VEL
LIN {X 0,Y 349.8,Z 365.483,A -85,B 0,C 180,E1 -13784.843,E2 -13784.843} C_VEL
LIN {X 0,Y 350.956,Z 355.922,A -85,B 0,C 180,E1 -13786.282,E2 -13786.282} C_VEL
LIN {X 0,Y 352.253,Z 345.351,A -85,B 0,C 180,E1 -13787.564,E2 -13787.564} C_VEL
LIN {X 0,Y 353.589,Z 333.6,A -85,B 0,C 180,E1 -13788.694,E2 -13788.694} C_VEL
LIN {X 0,Y 354.804,Z 322.182,A -85,B 0,C 180,E1 -13789.528,E2 -13789.528} C_VEL
LIN {X 0,Y 355.648,Z 310.185,A -85,B 0,C 180,E1 -13790.194,E2 -13790.194} C_VEL
LIN {X 0,Y 356.442,Z 297.307,A -85,B 0,C 180,E1 -13790.675,E2 -13790.675} C_VEL
LIN {X 0,Y 357.915,Z 223.737,A -85,B 0,C 180,E1 -13792.28,E2 -13792.28} C_VEL
LIN {X 0,Y 354.357,Z 201.945,A -85,B 0,C 180,E1 -13793.053,E2 -13793.053} C_VEL
LIN {X 0,Y 351.593,Z 188.339,A -85,B 0,C 180,E1 -13793.604,E2 -13793.604} C_VEL
LIN {X 0,Y 352.278,Z 182.206,A -85,B 0,C 180,E1 -13795.077,E2 -13795.077} C_VEL
LIN {X 0,Y 350.751,Z 173.389,A -85,B 0,C 180,E1 -13797.442,E2 -13797.442} C_VEL
LIN {X 0,Y 348.264,Z 162.143,A -85,B 0,C 180,E1 -13800.634,E2 -13800.634} C_VEL
LIN {X 0,Y 347.754,Z 160.174,A -85,B 0,C 180,E1 -13801.275,E2 -13801.275} C_VEL
LIN {X 0,Y 347.744,Z 160.172,A -85,B 0,C 180,E1 -13804.464,E2 -13804.464} C_VEL
LIN {X 0,Y 347.762,Z 160.166,A -85,B 0,C 180,E1 -13807.986,E2 -13807.986} C_VEL
LIN {X 0,Y 347.741,Z 160.168,A -85,B 0,C 180,E1 -13811.832,E2 -13811.832} C_VEL
LIN {X 0,Y 347.702,Z 160.175,A -85,B 0,C 180,E1 -13815.028,E2 -13815.028} C_VEL
LIN {X 0,Y 347.739,Z 160.169,A -85,B 0,C 180,E1 -13818.4,E2 -13818.4} C_VEL
LIN {X 0,Y 347.763,Z 160.165,A -85,B 0,C 180,E1 -13822.014,E2 -13822.014} C_VEL
LIN {X 0,Y 347.745,Z 160.166,A -85,B 0,C 180,E1 -13825.536,E2 -13825.536} C_VEL
LIN {X 0,Y 347.746,Z 160.165,A -85,B 0,C 180,E1 -13828.3,E2 -13828.3} C_VEL
LIN {X 0,Y 347.743,Z 160.161,A -85,B 0,C 180,E1 -13830.984,E2 -13830.984} C_VEL
LIN {X 0,Y 347.734,Z 160.166,A -85,B 0,C 180,E1 -13833.6,E2 -13833.6} C_VEL
LIN {X 0,Y 347.75,Z 160.161,A -85,B 0,C 180,E1 -13836.159,E2 -13836.159} C_VEL
LIN {X 0,Y 347.742,Z 160.157,A -85,B 0,C 180,E1 -13839.905,E2 -13839.905} C_VEL
LIN {X 0,Y 347.806,Z 160.162,A -85,B 0,C 180,E1 -13842.356,E2 -13842.356} C_VEL
LIN {X 0,Y 347.854,Z 160.152,A -85,B 0,C 180,E1 -13845.969,E2 -13845.969} C_VEL
LIN {X 0,Y 347.891,Z 160.139,A -85,B 0,C 180,E1 -13849.524,E2 -13849.524} C_VEL
LIN {X 0,Y 348.047,Z 160.129,A -85,B 0,C 180,E1 -13851.874,E2 -13851.874} C_VEL
LIN {X 0,Y 348.039,Z 160.122,A -85,B 0,C 180,E1 -13854.205,E2 -13854.205} C_VEL
LIN {X 0,Y 348.184,Z 160.104,A -85,B 0,C 180,E1 -13857.686,E2 -13857.686} C_VEL
LIN {X 0,Y 348.12,Z 160.116,A -85,B 0,C 180,E1 -13861.157,E2 -13861.157} C_VEL
LIN {X 0,Y 348.184,Z 160.107,A -85,B 0,C 180,E1 -13862.314,E2 -13862.314} C_VEL
LIN {X 0,Y 348.056,Z 160.127,A -85,B 0,C 180,E1 -13866.959,E2 -13866.959} C_VEL
LIN {X 0,Y 347.895,Z 160.15,A -85,B 0,C 180,E1 -13870.475,E2 -13870.475} C_VEL
LIN {X 0,Y 347.883,Z 160.153,A -85,B 0,C 180,E1 -13874.137,E2 -13874.137} C_VEL
LIN {X 0,Y 347.796,Z 160.16,A -85,B 0,C 180,E1 -13878.241,E2 -13878.241} C_VEL
LIN {X 0,Y 347.767,Z 160.169,A -85,B 0,C 180,E1 -13881.625,E2 -13881.625} C_VEL
LIN {X 0,Y 347.74,Z 160.173,A -85,B 0,C 180,E1 -13885.114,E2 -13885.114} C_VEL
LIN {X 0,Y 347.731,Z 160.174,A -85,B 0,C 180,E1 -13887.701,E2 -13887.701} C_VEL
LIN {X 0,Y 347.794,Z 160.267,A -85,B 0,C 180,E1 -13890.848,E2 -13890.848} C_VEL
LIN {X 0,Y 350.41,Z 171.924,A -85,B 0,C 180,E1 -13894.338,E2 -13894.338} C_VEL
LIN {X 0,Y 355.445,Z 184.83,A -85,B 0,C 180,E1 -13895.074,E2 -13895.074} C_VEL
LIN {X 0,Y 358.605,Z 199.918,A -85,B 0,C 180,E1 -13895.665,E2 -13895.665} C_VEL
LIN {X 0,Y 356.628,Z 280.32,A -85,B 0,C 180,E1 -13897.403,E2 -13897.403} C_VEL
LIN {X 0,Y 355.915,Z 294.018,A -85,B 0,C 180,E1 -13897.943,E2 -13897.943} C_VEL
LIN {X 0,Y 355.115,Z 306.661,A -85,B 0,C 180,E1 -13898.693,E2 -13898.693} C_VEL
LIN {X 0,Y 354.125,Z 317.28,A -85,B 0,C 180,E1 -13899.522,E2 -13899.522} C_VEL
LIN {X 0,Y 352.917,Z 328.194,A -85,B 0,C 180,E1 -13900.604,E2 -13900.604} C_VEL
LIN {X 0,Y 351.697,Z 338.575,A -85,B 0,C 180,E1 -13901.894,E2 -13901.894} C_VEL
LIN {X 0,Y 350.497,Z 347.942,A -85,B 0,C 180,E1 -13903.338,E2 -13903.338} C_VEL
LIN {X 0,Y 349.329,Z 356.484,A -85,B 0,C 180,E1 -13904.973,E2 -13904.973} C_VEL
LIN {X 0,Y 348.336,Z 363.71,A -85,B 0,C 180,E1 -13906.687,E2 -13906.687} C_VEL
LIN {X 0,Y 347.562,Z 369.596,A -85,B 0,C 180,E1 -13908.433,E2 -13908.433} C_VEL
LIN {X 0,Y 346.944,Z 374.592,A -85,B 0,C 180,E1 -13910.333,E2 -13910.333} C_VEL
LIN {X 0,Y 346.461,Z 378.7,A -85,B 0,C 180,E1 -13912.515,E2 -13912.515} C_VEL
LIN {X 0,Y 346.115,Z 380.957,A -85,B 0,C 180,E1 -13914.313,E2 -13914.313} C_VEL
LIN {X 0,Y 345.9,Z 382.35,A -85,B 0,C 180,E1 -13916.413,E2 -13916.413} C_VEL
LIN {X 0,Y 345.9,Z 382.44,A -85,B 0,C 180,E1 -13918.579,E2 -13918.579} C_VEL
LIN {X 0,Y 346.015,Z 380.993,A -85,B 0,C 180,E1 -13920.855,E2 -13920.855} C_VEL
LIN {X 0,Y 346.179,Z 379.481,A -85,B 0,C 180,E1 -13922.164,E2 -13922.164} C_VEL
LIN {X 0,Y 346.495,Z 376.14,A -85,B 0,C 180,E1 -13924.145,E2 -13924.145} C_VEL
LIN {X 0,Y 346.906,Z 371.496,A -85,B 0,C 180,E1 -13926.097,E2 -13926.097} C_VEL
LIN {X 0,Y 347.482,Z 365.664,A -85,B 0,C 180,E1 -13927.968,E2 -13927.968} C_VEL
LIN {X 0,Y 348.167,Z 359.185,A -85,B 0,C 180,E1 -13929.622,E2 -13929.622} C_VEL
LIN {X 0,Y 349.055,Z 351.545,A -85,B 0,C 180,E1 -13931.207,E2 -13931.207} C_VEL
LIN {X 0,Y 350.042,Z 342.213,A -85,B 0,C 180,E1 -13932.774,E2 -13932.774} C_VEL
LIN {X 0,Y 351.051,Z 332.349,A -85,B 0,C 180,E1 -13934.11,E2 -13934.11} C_VEL
LIN {X 0,Y 352.076,Z 321.871,A -85,B 0,C 180,E1 -13935.255,E2 -13935.255} C_VEL
LIN {X 0,Y 353.031,Z 309.996,A -85,B 0,C 180,E1 -13936.282,E2 -13936.282} C_VEL
LIN {X 0,Y 353.747,Z 297.913,A -85,B 0,C 180,E1 -13937.071,E2 -13937.071} C_VEL
LIN {X 0,Y 354.493,Z 284.279,A -85,B 0,C 180,E1 -13937.694,E2 -13937.694} C_VEL
LIN {X 0,Y 354.943,Z 270.261,A -85,B 0,C 180,E1 -13938.073,E2 -13938.073} C_VEL
LIN {X 0,Y 356.328,Z 198.601,A -85,B 0,C 180,E1 -13939.576,E2 -13939.576} C_VEL
LIN {X 0,Y 352.091,Z 177.388,A -85,B 0,C 180,E1 -13940.299,E2 -13940.299} C_VEL
LIN {X 0,Y 350.1,Z 171.43,A -85,B 0,C 180,E1 -13940.566,E2 -13940.566} C_VEL
LIN {X 0,Y 348.055,Z 160.132,A -85,B 0,C 180,E1 -13943.842,E2 -13943.842} C_VEL
LIN {X 0,Y 348.204,Z 160.108,A -85,B 0,C 180,E1 -13947.686,E2 -13947.686} C_VEL
LIN {X 0,Y 348.143,Z 160.116,A -85,B 0,C 180,E1 -13951.157,E2 -13951.157} C_VEL
LIN {X 0,Y 348.191,Z 160.116,A -85,B 0,C 180,E1 -13952.314,E2 -13952.314} C_VEL
LIN {X 0,Y 348.057,Z 160.127,A -85,B 0,C 180,E1 -13956.959,E2 -13956.959} C_VEL
LIN {X 0,Y 347.929,Z 160.145,A -85,B 0,C 180,E1 -13960.474,E2 -13960.474} C_VEL
LIN {X 0,Y 347.882,Z 160.153,A -85,B 0,C 180,E1 -13964.137,E2 -13964.137} C_VEL
LIN {X 0,Y 347.831,Z 160.157,A -85,B 0,C 180,E1 -13968.259,E2 -13968.259} C_VEL
LIN {X 0,Y 347.77,Z 160.162,A -85,B 0,C 180,E1 -13970.94,E2 -13970.94} C_VEL
LIN {X 0,Y 347.108,Z 160.25,A -85,B 0,C 180,E1 -13971.907,E2 -13971.907} C_VEL
LIN {X 0,Y 344.231,Z 160.61,A -85,B 0,C 180,E1 -13973.479,E2 -13973.479} C_VEL
LIN {X 0,Y 341.791,Z 160.914,A -85,B 0,C 180,E1 -13974.752,E2 -13974.752} C_VEL
LIN {X 0,Y 340.751,Z 161.042,A -85,B 0,C 180,E1 -13975.737,E2 -13975.737} C_VEL
LIN {X 0,Y 340.67,Z 161.048,A -85,B 0,C 180,E1 -13976.071,E2 -13976.071} C_VEL
LIN {X 0,Y 340.723,Z 161.043,A -85,B 0,C 180,E1 -13979.966,E2 -13979.966} C_VEL
LIN {X 0,Y 340.695,Z 161.046,A -85,B 0,C 180,E1 -13983.847,E2 -13983.847} C_VEL
LIN {X 0,Y 340.704,Z 161.043,A -85,B 0,C 180,E1 -13986.742,E2 -13986.742} C_VEL
LIN {X 0,Y 340.653,Z 161.049,A -85,B 0,C 180,E1 -13990.24,E2 -13990.24} C_VEL
LIN {X 0,Y 340.676,Z 161.048,A -85,B 0,C 180,E1 -13992.905,E2 -13992.905} C_VEL
LIN {X 0,Y 340.675,Z 161.05,A -85,B 0,C 180,E1 -13997.095,E2 -13997.095} C_VEL
LIN {X 0,Y 340.657,Z 161.048,A -85,B 0,C 180,E1 -14000.241,E2 -14000.241} C_VEL
LIN {X 0,Y 340.71,Z 161.043,A -85,B 0,C 180,E1 -14003.56,E2 -14003.56} C_VEL
LIN {X 0,Y 340.695,Z 161.043,A -85,B 0,C 180,E1 -14006.153,E2 -14006.153} C_VEL
LIN {X 0,Y 340.724,Z 161.04,A -85,B 0,C 180,E1 -14010.035,E2 -14010.035} C_VEL
LIN {X 0,Y 340.722,Z 161.044,A -85,B 0,C 180,E1 -14013.013,E2 -14013.013} C_VEL
LIN {X 0,Y 340.742,Z 161.038,A -85,B 0,C 180,E1 -14015.637,E2 -14015.637} C_VEL
LIN {X 0,Y 340.717,Z 161.041,A -85,B 0,C 180,E1 -14019.472,E2 -14019.472} C_VEL
LIN {X 0,Y 340.764,Z 161.036,A -85,B 0,C 180,E1 -14021.979,E2 -14021.979} C_VEL
LIN {X 0,Y 340.835,Z 161.026,A -85,B 0,C 180,E1 -14025.73,E2 -14025.73} C_VEL
LIN {X 0,Y 340.851,Z 161.024,A -85,B 0,C 180,E1 -14029.305,E2 -14029.305} C_VEL
LIN {X 0,Y 341.005,Z 161.006,A -85,B 0,C 180,E1 -14032.897,E2 -14032.897} C_VEL
LIN {X 0,Y 340.814,Z 161.028,A -85,B 0,C 180,E1 -14035.269,E2 -14035.269} C_VEL
LIN {X 0,Y 341.128,Z 160.99,A -85,B 0,C 180,E1 -14037.638,E2 -14037.638} C_VEL
LIN {X 0,Y 341.091,Z 160.994,A -85,B 0,C 180,E1 -14041.181,E2 -14041.181} C_VEL
LIN {X 0,Y 341.127,Z 160.993,A -85,B 0,C 180,E1 -14042.361,E2 -14042.361} C_VEL
LIN {X 0,Y 341.011,Z 161.004,A -85,B 0,C 180,E1 -14047.103,E2 -14047.103} C_VEL
LIN {X 0,Y 340.844,Z 161.025,A -85,B 0,C 180,E1 -14050.695,E2 -14050.695} C_VEL
LIN {X 0,Y 340.813,Z 161.03,A -85,B 0,C 180,E1 -14054.327,E2 -14054.327} C_VEL
LIN {X 0,Y 340.753,Z 161.037,A -85,B 0,C 180,E1 -14058.422,E2 -14058.422} C_VEL
LIN {X 0,Y 340.721,Z 161.044,A -85,B 0,C 180,E1 -14061.841,E2 -14061.841} C_VEL
LIN {X 0,Y 340.706,Z 161.042,A -85,B 0,C 180,E1 -14064.82,E2 -14064.82} C_VEL
LIN {X 0,Y 340.677,Z 161.046,A -85,B 0,C 180,E1 -14068.325,E2 -14068.325} C_VEL
LIN {X 0,Y 340.694,Z 161.046,A -85,B 0,C 180,E1 -14071.045,E2 -14071.045} C_VEL
LIN {X 0,Y 340.717,Z 161.046,A -85,B 0,C 180,E1 -14075.279,E2 -14075.279} C_VEL
LIN {X 0,Y 340.695,Z 161.043,A -85,B 0,C 180,E1 -14078.382,E2 -14078.382} C_VEL
LIN {X 0,Y 340.692,Z 161.044,A -85,B 0,C 180,E1 -14082.044,E2 -14082.044} C_VEL
LIN {X 0,Y 340.651,Z 161.049,A -85,B 0,C 180,E1 -14086.227,E2 -14086.227} C_VEL
LIN {X 0,Y 340.67,Z 161.049,A -85,B 0,C 180,E1 -14088.688,E2 -14088.688} C_VEL
LIN {X 0,Y 340.719,Z 161.04,A -85,B 0,C 180,E1 -14091.77,E2 -14091.77} C_VEL
LIN {X 0,Y 340.723,Z 161.04,A -85,B 0,C 180,E1 -14095.596,E2 -14095.596} C_VEL
LIN {X 0,Y 340.777,Z 161.227,A -85,B 0,C 180,E1 -14099.691,E2 -14099.691} C_VEL
LIN {X 0,Y 343.338,Z 174.082,A -85,B 0,C 180,E1 -14103.235,E2 -14103.235} C_VEL
LIN {X 0,Y 344.513,Z 180.546,A -85,B 0,C 180,E1 -14104.957,E2 -14104.957} C_VEL
LIN {X 0,Y 343.748,Z 189.165,A -85,B 0,C 180,E1 -14107.076,E2 -14107.076} C_VEL
LIN {X 0,Y 349.253,Z 225.014,A -85,B 0,C 180,E1 -14108.235,E2 -14108.235} C_VEL
LIN {X 0,Y 347.743,Z 298.036,A -85,B 0,C 180,E1 -14109.828,E2 -14109.828} C_VEL
LIN {X 0,Y 347.047,Z 311.669,A -85,B 0,C 180,E1 -14110.364,E2 -14110.364} C_VEL
LIN {X 0,Y 346.088,Z 324.533,A -85,B 0,C 180,E1 -14111.116,E2 -14111.116} C_VEL
LIN {X 0,Y 345.01,Z 336.302,A -85,B 0,C 180,E1 -14112.055,E2 -14112.055} C_VEL
LIN {X 0,Y 343.852,Z 347.675,A -85,B 0,C 180,E1 -14113.22,E2 -14113.22} C_VEL
LIN {X 0,Y 342.805,Z 357.936,A -85,B 0,C 180,E1 -14114.543,E2 -14114.543} C_VEL
LIN {X 0,Y 341.782,Z 367.157,A -85,B 0,C 180,E1 -14116.018,E2 -14116.018} C_VEL
LIN {X 0,Y 340.943,Z 374.769,A -85,B 0,C 180,E1 -14117.5,E2 -14117.5} C_VEL
LIN {X 0,Y 340.132,Z 382.229,A -85,B 0,C 180,E1 -14119.283,E2 -14119.283} C_VEL
LIN {X 0,Y 339.602,Z 388.208,A -85,B 0,C 180,E1 -14121.071,E2 -14121.071} C_VEL
LIN {X 0,Y 339.269,Z 392.913,A -85,B 0,C 180,E1 -14122.86,E2 -14122.86} C_VEL
LIN {X 0,Y 339.129,Z 395.532,A -85,B 0,C 180,E1 -14124.121,E2 -14124.121} C_VEL
LIN {X 0,Y 339.07,Z 399.028,A -85,B 0,C 180,E1 -14126.435,E2 -14126.435} C_VEL
LIN {X 0,Y 338.999,Z 400.204,A -85,B 0,C 180,E1 -14127.624,E2 -14127.624} C_VEL
LIN {X 0,Y 339.019,Z 400.931,A -85,B 0,C 180,E1 -14128.812,E2 -14128.812} C_VEL
LIN {X 0,Y 339.067,Z 401.264,A -85,B 0,C 180,E1 -14130,E2 -14130} C_VEL
LIN {X 0,Y 339.006,Z 401.201,A -85,B 0,C 180,E1 -14131.188,E2 -14131.188} C_VEL
LIN {X 0,Y 338.997,Z 400.74,A -85,B 0,C 180,E1 -14132.376,E2 -14132.376} C_VEL
LIN {X 0,Y 339.064,Z 399.839,A -85,B 0,C 180,E1 -14133.565,E2 -14133.565} C_VEL
LIN {X 0,Y 339.111,Z 396.976,A -85,B 0,C 180,E1 -14135.85,E2 -14135.85} C_VEL
LIN {X 0,Y 339.398,Z 393.399,A -85,B 0,C 180,E1 -14137.735,E2 -14137.735} C_VEL
LIN {X 0,Y 339.823,Z 388.894,A -85,B 0,C 180,E1 -14139.524,E2 -14139.524} C_VEL
LIN {X 0,Y 340.507,Z 383.188,A -85,B 0,C 180,E1 -14141.308,E2 -14141.308} C_VEL
LIN {X 0,Y 341.488,Z 376.06,A -85,B 0,C 180,E1 -14143.085,E2 -14143.085} C_VEL
LIN {X 0,Y 342.75,Z 367.189,A -85,B 0,C 180,E1 -14144.851,E2 -14144.851} C_VEL
LIN {X 0,Y 344,Z 357.286,A -85,B 0,C 180,E1 -14146.445,E2 -14146.445} C_VEL
LIN {X 0,Y 345.356,Z 346.873,A -85,B 0,C 180,E1 -14147.773,E2 -14147.773} C_VEL
LIN {X 0,Y 346.695,Z 335.535,A -85,B 0,C 180,E1 -14148.926,E2 -14148.926} C_VEL
LIN {X 0,Y 348.013,Z 323.796,A -85,B 0,C 180,E1 -14149.848,E2 -14149.848} C_VEL
LIN {X 0,Y 349.014,Z 310.992,A -85,B 0,C 180,E1 -14150.595,E2 -14150.595} C_VEL
LIN {X 0,Y 349.908,Z 297.497,A -85,B 0,C 180,E1 -14151.118,E2 -14151.118} C_VEL
LIN {X 0,Y 351.54,Z 225.178,A -85,B 0,C 180,E1 -14152.723,E2 -14152.723} C_VEL
LIN {X 0,Y 348.082,Z 203.705,A -85,B 0,C 180,E1 -14153.507,E2 -14153.507} C_VEL
LIN {X 0,Y 344.893,Z 188.079,A -85,B 0,C 180,E1 -14154.171,E2 -14154.171} C_VEL
LIN {X 0,Y 345.402,Z 183.511,A -85,B 0,C 180,E1 -14155.296,E2 -14155.296} C_VEL
LIN {X 0,Y 343.831,Z 174.731,A -85,B 0,C 180,E1 -14157.712,E2 -14157.712} C_VEL
LIN {X 0,Y 341.323,Z 163.526,A -85,B 0,C 180,E1 -14160.982,E2 -14160.982} C_VEL
LIN {X 0,Y 340.722,Z 161.052,A -85,B 0,C 180,E1 -14161.735,E2 -14161.735} C_VEL
LIN {X 0,Y 340.716,Z 161.046,A -85,B 0,C 180,E1 -14165.279,E2 -14165.279} C_VEL
LIN {X 0,Y 340.694,Z 161.047,A -85,B 0,C 180,E1 -14168.382,E2 -14168.382} C_VEL
LIN {X 0,Y 340.692,Z 161.046,A -85,B 0,C 180,E1 -14172.044,E2 -14172.044} C_VEL
LIN {X 0,Y 340.651,Z 161.054,A -85,B 0,C 180,E1 -14176.228,E2 -14176.228} C_VEL
LIN {X 0,Y 340.67,Z 161.052,A -85,B 0,C 180,E1 -14178.688,E2 -14178.688} C_VEL
LIN {X 0,Y 340.719,Z 161.043,A -85,B 0,C 180,E1 -14181.771,E2 -14181.771} C_VEL
LIN {X 0,Y 340.724,Z 161.041,A -85,B 0,C 180,E1 -14185.596,E2 -14185.596} C_VEL
LIN {X 0,Y 340.694,Z 161.047,A -85,B 0,C 180,E1 -14188.955,E2 -14188.955} C_VEL
LIN {X 0,Y 340.711,Z 161.044,A -85,B 0,C 180,E1 -14193.012,E2 -14193.012} C_VEL
LIN {X 0,Y 340.702,Z 161.046,A -85,B 0,C 180,E1 -14196.925,E2 -14196.925} C_VEL
LIN {X 0,Y 340.694,Z 161.042,A -85,B 0,C 180,E1 -14200.728,E2 -14200.728} C_VEL
LIN {X 0,Y 340.726,Z 161.037,A -85,B 0,C 180,E1 -14203.216,E2 -14203.216} C_VEL
LIN {X 0,Y 340.818,Z 161.03,A -85,B 0,C 180,E1 -14206.889,E2 -14206.889} C_VEL
LIN {X 0,Y 340.882,Z 161.021,A -85,B 0,C 180,E1 -14210.506,E2 -14210.506} C_VEL
LIN {X 0,Y 341.016,Z 160.995,A -85,B 0,C 180,E1 -14212.897,E2 -14212.897} C_VEL
LIN {X 0,Y 340.81,Z 161.028,A -85,B 0,C 180,E1 -14215.269,E2 -14215.269} C_VEL
LIN {X 0,Y 341.121,Z 160.983,A -85,B 0,C 180,E1 -14217.638,E2 -14217.638} C_VEL
LIN {X 0,Y 341.091,Z 160.991,A -85,B 0,C 180,E1 -14221.181,E2 -14221.181} C_VEL
LIN {X 0,Y 341.121,Z 160.987,A -85,B 0,C 180,E1 -14222.362,E2 -14222.362} C_VEL
LIN {X 0,Y 340.991,Z 161.003,A -85,B 0,C 180,E1 -14226.479,E2 -14226.479} C_VEL
LIN {X 0,Y 340.884,Z 161.018,A -85,B 0,C 180,E1 -14229.494,E2 -14229.494} C_VEL
LIN {X 0,Y 340.844,Z 161.024,A -85,B 0,C 180,E1 -14233.11,E2 -14233.11} C_VEL
LIN {X 0,Y 340.737,Z 161.041,A -85,B 0,C 180,E1 -14236.784,E2 -14236.784} C_VEL
LIN {X 0,Y 340.695,Z 161.047,A -85,B 0,C 180,E1 -14239.272,E2 -14239.272} C_VEL
LIN {X 0,Y 340.704,Z 161.046,A -85,B 0,C 180,E1 -14243.075,E2 -14243.075} C_VEL
LIN {X 0,Y 340.713,Z 161.049,A -85,B 0,C 180,E1 -14246.988,E2 -14246.988} C_VEL
LIN {X 0,Y 340.76,Z 161.237,A -85,B 0,C 180,E1 -14250.365,E2 -14250.365} C_VEL
LIN {X 0,Y 343.268,Z 172.141,A -85,B 0,C 180,E1 -14253.735,E2 -14253.735} C_VEL
LIN {X 0,Y 349.402,Z 187.486,A -85,B 0,C 180,E1 -14254.653,E2 -14254.653} C_VEL
LIN {X 0,Y 352.18,Z 201.551,A -85,B 0,C 180,E1 -14255.212,E2 -14255.212} C_VEL
LIN {X 0,Y 350.154,Z 279.576,A -85,B 0,C 180,E1 -14256.919,E2 -14256.919} C_VEL
LIN {X 0,Y 349.434,Z 293.316,A -85,B 0,C 180,E1 -14257.456,E2 -14257.456} C_VEL
LIN {X 0,Y 348.631,Z 305.531,A -85,B 0,C 180,E1 -14258.168,E2 -14258.168} C_VEL
LIN {X 0,Y 347.612,Z 316.418,A -85,B 0,C 180,E1 -14259.008,E2 -14259.008} C_VEL
LIN {X 0,Y 346.291,Z 327.963,A -85,B 0,C 180,E1 -14260.156,E2 -14260.156} C_VEL
LIN {X 0,Y 345.009,Z 338.458,A -85,B 0,C 180,E1 -14261.476,E2 -14261.476} C_VEL
LIN {X 0,Y 343.669,Z 348.319,A -85,B 0,C 180,E1 -14263.022,E2 -14263.022} C_VEL
LIN {X 0,Y 342.539,Z 356.171,A -85,B 0,C 180,E1 -14264.546,E2 -14264.546} C_VEL
LIN {X 0,Y 341.439,Z 363.625,A -85,B 0,C 180,E1 -14266.331,E2 -14266.331} C_VEL
LIN {X 0,Y 340.678,Z 369.094,A -85,B 0,C 180,E1 -14267.959,E2 -14267.959} C_VEL
LIN {X 0,Y 339.913,Z 374.809,A -85,B 0,C 180,E1 -14270.137,E2 -14270.137} C_VEL
LIN {X 0,Y 339.489,Z 378.165,A -85,B 0,C 180,E1 -14271.875,E2 -14271.875} C_VEL
LIN {X 0,Y 339.083,Z 380.915,A -85,B 0,C 180,E1 -14273.934,E2 -14273.934} C_VEL
LIN {X 0,Y 338.843,Z 382.441,A -85,B 0,C 180,E1 -14276.063,E2 -14276.063} C_VEL
LIN {X 0,Y 338.776,Z 382.682,A -85,B 0,C 180,E1 -14278.273,E2 -14278.273} C_VEL
LIN {X 0,Y 338.896,Z 381.47,A -85,B 0,C 180,E1 -14280.575,E2 -14280.575} C_VEL
LIN {X 0,Y 339.208,Z 378.677,A -85,B 0,C 180,E1 -14282.882,E2 -14282.882} C_VEL
LIN {X 0,Y 339.57,Z 374.92,A -85,B 0,C 180,E1 -14284.895,E2 -14284.895} C_VEL
LIN {X 0,Y 340.066,Z 369.85,A -85,B 0,C 180,E1 -14286.879,E2 -14286.879} C_VEL
LIN {X 0,Y 340.701,Z 363.163,A -85,B 0,C 180,E1 -14288.872,E2 -14288.872} C_VEL
LIN {X 0,Y 341.668,Z 354.997,A -85,B 0,C 180,E1 -14290.785,E2 -14290.785} C_VEL
LIN {X 0,Y 342.696,Z 346.347,A -85,B 0,C 180,E1 -14292.392,E2 -14292.392} C_VEL
LIN {X 0,Y 343.771,Z 336.198,A -85,B 0,C 180,E1 -14293.918,E2 -14293.918} C_VEL
LIN {X 0,Y 344.989,Z 325.074,A -85,B 0,C 180,E1 -14295.247,E2 -14295.247} C_VEL
LIN {X 0,Y 345.873,Z 314.109,A -85,B 0,C 180,E1 -14296.286,E2 -14296.286} C_VEL
LIN {X 0,Y 346.811,Z 301.624,A -85,B 0,C 180,E1 -14297.194,E2 -14297.194} C_VEL
LIN {X 0,Y 347.573,Z 289.111,A -85,B 0,C 180,E1 -14297.853,E2 -14297.853} C_VEL
LIN {X 0,Y 348.062,Z 276.124,A -85,B 0,C 180,E1 -14298.295,E2 -14298.295} C_VEL
LIN {X 0,Y 349.586,Z 199.418,A -85,B 0,C 180,E1 -14299.949,E2 -14299.949} C_VEL
LIN {X 0,Y 345.669,Z 179.662,A -85,B 0,C 180,E1 -14300.639,E2 -14300.639} C_VEL
LIN {X 0,Y 342.947,Z 171.606,A -85,B 0,C 180,E1 -14301.01,E2 -14301.01} C_VEL
LIN {X 0,Y 341.017,Z 161.008,A -85,B 0,C 180,E1 -14304.16,E2 -14304.16} C_VEL
LIN {X 0,Y 341.166,Z 160.985,A -85,B 0,C 180,E1 -14307.639,E2 -14307.639} C_VEL
LIN {X 0,Y 341.112,Z 160.992,A -85,B 0,C 180,E1 -14311.181,E2 -14311.181} C_VEL
LIN {X 0,Y 341.128,Z 160.995,A -85,B 0,C 180,E1 -14312.362,E2 -14312.362} C_VEL
LIN {X 0,Y 341.017,Z 161.006,A -85,B 0,C 180,E1 -14315.915,E2 -14315.915} C_VEL
LIN {X 0,Y 340.913,Z 161.017,A -85,B 0,C 180,E1 -14319.493,E2 -14319.493} C_VEL
LIN {X 0,Y 340.845,Z 161.025,A -85,B 0,C 180,E1 -14323.11,E2 -14323.11} C_VEL
LIN {X 0,Y 340.752,Z 161.036,A -85,B 0,C 180,E1 -14326.783,E2 -14326.783} C_VEL
LIN {X 0,Y 340.76,Z 161.036,A -85,B 0,C 180,E1 -14329.268,E2 -14329.268} C_VEL
LIN {X 0,Y 340.703,Z 161.043,A -85,B 0,C 180,E1 -14333.075,E2 -14333.075} C_VEL
LIN {X 0,Y 340.67,Z 161.048,A -85,B 0,C 180,E1 -14336.071,E2 -14336.071} C_VEL
LIN {X 0,Y 340.011,Z 161.13,A -85,B 0,C 180,E1 -14337.058,E2 -14337.058} C_VEL
LIN {X 0,Y 337.154,Z 161.484,A -85,B 0,C 180,E1 -14338.663,E2 -14338.663} C_VEL
LIN {X 0,Y 334.732,Z 161.789,A -85,B 0,C 180,E1 -14339.962,E2 -14339.962} C_VEL
LIN {X 0,Y 333.698,Z 161.915,A -85,B 0,C 180,E1 -14340.968,E2 -14340.968} C_VEL
LIN {X 0,Y 333.618,Z 161.924,A -85,B 0,C 180,E1 -14341.309,E2 -14341.309} C_VEL
LIN {X 0,Y 333.687,Z 161.916,A -85,B 0,C 180,E1 -14344.774,E2 -14344.774} C_VEL
LIN {X 0,Y 333.645,Z 161.925,A -85,B 0,C 180,E1 -14347.652,E2 -14347.652} C_VEL
LIN {X 0,Y 333.605,Z 161.927,A -85,B 0,C 180,E1 -14350.774,E2 -14350.774} C_VEL
LIN {X 0,Y 333.593,Z 161.927,A -85,B 0,C 180,E1 -14354.25,E2 -14354.25} C_VEL
LIN {X 0,Y 333.64,Z 161.923,A -85,B 0,C 180,E1 -14357.618,E2 -14357.618} C_VEL
LIN {X 0,Y 333.636,Z 161.928,A -85,B 0,C 180,E1 -14361.206,E2 -14361.206} C_VEL
LIN {X 0,Y 333.676,Z 161.918,A -85,B 0,C 180,E1 -14363.861,E2 -14363.861} C_VEL
LIN {X 0,Y 333.646,Z 161.923,A -85,B 0,C 180,E1 -14367.413,E2 -14367.413} C_VEL
LIN {X 0,Y 333.656,Z 161.925,A -85,B 0,C 180,E1 -14371.022,E2 -14371.022} C_VEL
LIN {X 0,Y 333.699,Z 161.917,A -85,B 0,C 180,E1 -14375.088,E2 -14375.088} C_VEL
LIN {X 0,Y 333.657,Z 161.923,A -85,B 0,C 180,E1 -14379.018,E2 -14379.018} C_VEL
LIN {X 0,Y 333.716,Z 161.913,A -85,B 0,C 180,E1 -14381.585,E2 -14381.585} C_VEL
LIN {X 0,Y 333.777,Z 161.905,A -85,B 0,C 180,E1 -14385.6,E2 -14385.6} C_VEL
LIN {X 0,Y 333.82,Z 161.901,A -85,B 0,C 180,E1 -14389.078,E2 -14389.078} C_VEL
LIN {X 0,Y 333.96,Z 161.884,A -85,B 0,C 180,E1 -14392.746,E2 -14392.746} C_VEL
LIN {X 0,Y 333.781,Z 161.904,A -85,B 0,C 180,E1 -14395.169,E2 -14395.169} C_VEL
LIN {X 0,Y 334.069,Z 161.869,A -85,B 0,C 180,E1 -14397.588,E2 -14397.588} C_VEL
LIN {X 0,Y 334.062,Z 161.869,A -85,B 0,C 180,E1 -14401.205,E2 -14401.205} C_VEL
LIN {X 0,Y 334.068,Z 161.871,A -85,B 0,C 180,E1 -14402.411,E2 -14402.411} C_VEL
LIN {X 0,Y 333.991,Z 161.883,A -85,B 0,C 180,E1 -14406.039,E2 -14406.039} C_VEL
LIN {X 0,Y 333.916,Z 161.889,A -85,B 0,C 180,E1 -14408.472,E2 -14408.472} C_VEL
LIN {X 0,Y 333.776,Z 161.909,A -85,B 0,C 180,E1 -14412.155,E2 -14412.155} C_VEL
LIN {X 0,Y 333.736,Z 161.91,A -85,B 0,C 180,E1 -14414.638,E2 -14414.638} C_VEL
LIN {X 0,Y 333.692,Z 161.915,A -85,B 0,C 180,E1 -14418.6,E2 -14418.6} C_VEL
LIN {X 0,Y 333.651,Z 161.921,A -85,B 0,C 180,E1 -14422.281,E2 -14422.281} C_VEL
LIN {X 0,Y 333.658,Z 161.921,A -85,B 0,C 180,E1 -14425.077,E2 -14425.077} C_VEL
LIN {X 0,Y 333.63,Z 161.925,A -85,B 0,C 180,E1 -14428.98,E2 -14428.98} C_VEL
LIN {X 0,Y 333.645,Z 161.922,A -85,B 0,C 180,E1 -14432.587,E2 -14432.587} C_VEL
LIN {X 0,Y 333.675,Z 161.918,A -85,B 0,C 180,E1 -14436.139,E2 -14436.139} C_VEL
LIN {X 0,Y 333.621,Z 161.93,A -85,B 0,C 180,E1 -14439.196,E2 -14439.196} C_VEL
LIN {X 0,Y 333.628,Z 161.924,A -85,B 0,C 180,E1 -14442.499,E2 -14442.499} C_VEL
LIN {X 0,Y 333.595,Z 161.928,A -85,B 0,C 180,E1 -14445.954,E2 -14445.954} C_VEL
LIN {X 0,Y 333.603,Z 161.929,A -85,B 0,C 180,E1 -14449.324,E2 -14449.324} C_VEL
LIN {X 0,Y 333.662,Z 161.923,A -85,B 0,C 180,E1 -14453.169,E2 -14453.169} C_VEL
LIN {X 0,Y 333.674,Z 161.92,A -85,B 0,C 180,E1 -14455.341,E2 -14455.341} C_VEL
LIN {X 0,Y 333.707,Z 162.053,A -85,B 0,C 180,E1 -14459.333,E2 -14459.333} C_VEL
LIN {X 0,Y 336.074,Z 173.624,A -85,B 0,C 180,E1 -14462.608,E2 -14462.608} C_VEL
LIN {X 0,Y 337.519,Z 181.395,A -85,B 0,C 180,E1 -14464.731,E2 -14464.731} C_VEL
LIN {X 0,Y 337.174,Z 186.74,A -85,B 0,C 180,E1 -14466.083,E2 -14466.083} C_VEL
LIN {X 0,Y 336.886,Z 189.05,A -85,B 0,C 180,E1 -14466.648,E2 -14466.648} C_VEL
LIN {X 0,Y 342.516,Z 225.422,A -85,B 0,C 180,E1 -14467.849,E2 -14467.849} C_VEL
LIN {X 0,Y 340.992,Z 297.506,A -85,B 0,C 180,E1 -14469.452,E2 -14469.452} C_VEL
LIN {X 0,Y 340.318,Z 311.211,A -85,B 0,C 180,E1 -14469.999,E2 -14469.999} C_VEL
LIN {X 0,Y 339.38,Z 323.646,A -85,B 0,C 180,E1 -14470.729,E2 -14470.729} C_VEL
LIN {X 0,Y 338.241,Z 335.571,A -85,B 0,C 180,E1 -14471.683,E2 -14471.683} C_VEL
LIN {X 0,Y 337.041,Z 347.043,A -85,B 0,C 180,E1 -14472.87,E2 -14472.87} C_VEL
LIN {X 0,Y 335.886,Z 357.676,A -85,B 0,C 180,E1 -14474.258,E2 -14474.258} C_VEL
LIN {X 0,Y 334.852,Z 366.687,A -85,B 0,C 180,E1 -14475.723,E2 -14475.723} C_VEL
LIN {X 0,Y 333.959,Z 374.346,A -85,B 0,C 180,E1 -14477.234,E2 -14477.234} C_VEL
LIN {X 0,Y 333.097,Z 381.847,A -85,B 0,C 180,E1 -14479.054,E2 -14479.054} C_VEL
LIN {X 0,Y 332.559,Z 387.864,A -85,B 0,C 180,E1 -14480.88,E2 -14480.88} C_VEL
LIN {X 0,Y 332.195,Z 392.602,A -85,B 0,C 180,E1 -14482.707,E2 -14482.707} C_VEL
LIN {X 0,Y 332.028,Z 395.579,A -85,B 0,C 180,E1 -14484.18,E2 -14484.18} C_VEL
LIN {X 0,Y 331.995,Z 398.776,A -85,B 0,C 180,E1 -14486.359,E2 -14486.359} C_VEL
LIN {X 0,Y 331.917,Z 399.972,A -85,B 0,C 180,E1 -14487.573,E2 -14487.573} C_VEL
LIN {X 0,Y 331.924,Z 400.717,A -85,B 0,C 180,E1 -14488.787,E2 -14488.787} C_VEL
LIN {X 0,Y 331.97,Z 401.061,A -85,B 0,C 180,E1 -14490,E2 -14490} C_VEL
LIN {X 0,Y 331.912,Z 401.011,A -85,B 0,C 180,E1 -14491.213,E2 -14491.213} C_VEL
LIN {X 0,Y 331.914,Z 400.568,A -85,B 0,C 180,E1 -14492.427,E2 -14492.427} C_VEL
LIN {X 0,Y 331.967,Z 399.684,A -85,B 0,C 180,E1 -14493.641,E2 -14493.641} C_VEL
LIN {X 0,Y 332.005,Z 397.136,A -85,B 0,C 180,E1 -14495.781,E2 -14495.781} C_VEL
LIN {X 0,Y 332.355,Z 393.296,A -85,B 0,C 180,E1 -14497.9,E2 -14497.9} C_VEL
LIN {X 0,Y 332.798,Z 388.825,A -85,B 0,C 180,E1 -14499.726,E2 -14499.726} C_VEL
LIN {X 0,Y 333.506,Z 383.159,A -85,B 0,C 180,E1 -14501.548,E2 -14501.548} C_VEL
LIN {X 0,Y 334.56,Z 376.092,A -85,B 0,C 180,E1 -14503.36,E2 -14503.36} C_VEL
LIN {X 0,Y 335.871,Z 367.267,A -85,B 0,C 180,E1 -14505.163,E2 -14505.163} C_VEL
LIN {X 0,Y 337.17,Z 357.581,A -85,B 0,C 180,E1 -14506.762,E2 -14506.762} C_VEL
LIN {X 0,Y 338.611,Z 347.105,A -85,B 0,C 180,E1 -14508.14,E2 -14508.14} C_VEL
LIN {X 0,Y 340.015,Z 335.861,A -85,B 0,C 180,E1 -14509.312,E2 -14509.312} C_VEL
LIN {X 0,Y 341.246,Z 325.244,A -85,B 0,C 180,E1 -14510.18,E2 -14510.18} C_VEL
LIN {X 0,Y 342.33,Z 312.526,A -85,B 0,C 180,E1 -14510.977,E2 -14510.977} C_VEL
LIN {X 0,Y 343.306,Z 299.885,A -85,B 0,C 180,E1 -14511.504,E2 -14511.504} C_VEL
LIN {X 0,Y 343.833,Z 281.025,A -85,B 0,C 180,E1 -14511.984,E2 -14511.984} C_VEL
LIN {X 0,Y 345.085,Z 225.798,A -85,B 0,C 180,E1 -14513.216,E2 -14513.216} C_VEL
LIN {X 0,Y 341.66,Z 204.44,A -85,B 0,C 180,E1 -14514.025,E2 -14514.025} C_VEL
LIN {X 0,Y 338.208,Z 187.925,A -85,B 0,C 180,E1 -14514.742,E2 -14514.742} C_VEL
LIN {X 0,Y 338.51,Z 184.855,A -85,B 0,C 180,E1 -14515.519,E2 -14515.519} C_VEL
LIN {X 0,Y 336.917,Z 176.107,A -85,B 0,C 180,E1 -14517.992,E2 -14517.992} C_VEL
LIN {X 0,Y 334.63,Z 165.829,A -85,B 0,C 180,E1 -14521.059,E2 -14521.059} C_VEL
LIN {X 0,Y 333.666,Z 161.928,A -85,B 0,C 180,E1 -14522.334,E2 -14522.334} C_VEL
LIN {X 0,Y 333.674,Z 161.92,A -85,B 0,C 180,E1 -14526.14,E2 -14526.14} C_VEL
LIN {X 0,Y 333.621,Z 161.93,A -85,B 0,C 180,E1 -14529.196,E2 -14529.196} C_VEL
LIN {X 0,Y 333.628,Z 161.927,A -85,B 0,C 180,E1 -14532.499,E2 -14532.499} C_VEL
LIN {X 0,Y 333.595,Z 161.933,A -85,B 0,C 180,E1 -14535.955,E2 -14535.955} C_VEL
LIN {X 0,Y 333.603,Z 161.927,A -85,B 0,C 180,E1 -14539.325,E2 -14539.325} C_VEL
LIN {X 0,Y 333.663,Z 161.917,A -85,B 0,C 180,E1 -14543.169,E2 -14543.169} C_VEL
LIN {X 0,Y 333.675,Z 161.92,A -85,B 0,C 180,E1 -14545.341,E2 -14545.341} C_VEL
LIN {X 0,Y 333.63,Z 161.923,A -85,B 0,C 180,E1 -14548.222,E2 -14548.222} C_VEL
LIN {X 0,Y 333.63,Z 161.918,A -85,B 0,C 180,E1 -14551.02,E2 -14551.02} C_VEL
LIN {X 0,Y 333.657,Z 161.913,A -85,B 0,C 180,E1 -14554.923,E2 -14554.923} C_VEL
LIN {X 0,Y 333.641,Z 161.914,A -85,B 0,C 180,E1 -14559.017,E2 -14559.017} C_VEL
LIN {X 0,Y 333.712,Z 161.915,A -85,B 0,C 180,E1 -14561.585,E2 -14561.585} C_VEL
LIN {X 0,Y 333.762,Z 161.906,A -85,B 0,C 180,E1 -14565.611,E2 -14565.611} C_VEL
LIN {X 0,Y 333.812,Z 161.892,A -85,B 0,C 180,E1 -14569.077,E2 -14569.077} C_VEL
LIN {X 0,Y 333.972,Z 161.873,A -85,B 0,C 180,E1 -14572.746,E2 -14572.746} C_VEL
LIN {X 0,Y 333.777,Z 161.904,A -85,B 0,C 180,E1 -14575.169,E2 -14575.169} C_VEL
LIN {X 0,Y 334.061,Z 161.863,A -85,B 0,C 180,E1 -14577.589,E2 -14577.589} C_VEL
LIN {X 0,Y 334.061,Z 161.867,A -85,B 0,C 180,E1 -14581.206,E2 -14581.206} C_VEL
LIN {X 0,Y 334.062,Z 161.866,A -85,B 0,C 180,E1 -14582.412,E2 -14582.412} C_VEL
LIN {X 0,Y 333.961,Z 161.879,A -85,B 0,C 180,E1 -14586.471,E2 -14586.471} C_VEL
LIN {X 0,Y 333.822,Z 161.897,A -85,B 0,C 180,E1 -14589.696,E2 -14589.696} C_VEL
LIN {X 0,Y 333.789,Z 161.904,A -85,B 0,C 180,E1 -14593.392,E2 -14593.392} C_VEL
LIN {X 0,Y 333.683,Z 161.921,A -85,B 0,C 180,E1 -14597.15,E2 -14597.15} C_VEL
LIN {X 0,Y 333.638,Z 161.927,A -85,B 0,C 180,E1 -14599.697,E2 -14599.697} C_VEL
LIN {X 0,Y 333.652,Z 161.923,A -85,B 0,C 180,E1 -14602.281,E2 -14602.281} C_VEL
LIN {X 0,Y 333.661,Z 161.927,A -85,B 0,C 180,E1 -14605.078,E2 -14605.078} C_VEL
LIN {X 0,Y 333.654,Z 161.926,A -85,B 0,C 180,E1 -14608.978,E2 -14608.978} C_VEL
LIN {X 0,Y 333.695,Z 162.003,A -85,B 0,C 180,E1 -14609.79,E2 -14609.79} C_VEL
LIN {X 0,Y 335.989,Z 171.906,A -85,B 0,C 180,E1 -14612.946,E2 -14612.946} C_VEL
LIN {X 0,Y 336.155,Z 172.671,A -85,B 0,C 180,E1 -14613.134,E2 -14613.134} C_VEL
LIN {X 0,Y 343.212,Z 189.516,A -85,B 0,C 180,E1 -14614.183,E2 -14614.183} C_VEL
LIN {X 0,Y 345.73,Z 201.684,A -85,B 0,C 180,E1 -14614.694,E2 -14614.694} C_VEL
LIN {X 0,Y 343.651,Z 280.678,A -85,B 0,C 180,E1 -14616.477,E2 -14616.477} C_VEL
LIN {X 0,Y 342.848,Z 294.179,A -85,B 0,C 180,E1 -14617.024,E2 -14617.024} C_VEL
LIN {X 0,Y 342.026,Z 306.337,A -85,B 0,C 180,E1 -14617.76,E2 -14617.76} C_VEL
LIN {X 0,Y 340.919,Z 317.619,A -85,B 0,C 180,E1 -14618.667,E2 -14618.667} C_VEL
LIN {X 0,Y 339.551,Z 328.777,A -85,B 0,C 180,E1 -14619.812,E2 -14619.812} C_VEL
LIN {X 0,Y 338.239,Z 338.989,A -85,B 0,C 180,E1 -14621.13,E2 -14621.13} C_VEL
LIN {X 0,Y 336.887,Z 348.525,A -85,B 0,C 180,E1 -14622.661,E2 -14622.661} C_VEL
LIN {X 0,Y 335.67,Z 356.43,A -85,B 0,C 180,E1 -14624.225,E2 -14624.225} C_VEL
LIN {X 0,Y 334.479,Z 364.078,A -85,B 0,C 180,E1 -14626.101,E2 -14626.101} C_VEL
LIN {X 0,Y 333.572,Z 370.249,A -85,B 0,C 180,E1 -14628.014,E2 -14628.014} C_VEL
LIN {X 0,Y 332.853,Z 375.296,A -85,B 0,C 180,E1 -14630.057,E2 -14630.057} C_VEL
LIN {X 0,Y 332.321,Z 379.079,A -85,B 0,C 180,E1 -14632.171,E2 -14632.171} C_VEL
LIN {X 0,Y 332.033,Z 380.973,A -85,B 0,C 180,E1 -14633.653,E2 -14633.653} C_VEL
LIN {X 0,Y 331.766,Z 382.537,A -85,B 0,C 180,E1 -14635.707,E2 -14635.707} C_VEL
LIN {X 0,Y 331.667,Z 382.912,A -85,B 0,C 180,E1 -14638.011,E2 -14638.011} C_VEL
LIN {X 0,Y 331.777,Z 381.898,A -85,B 0,C 180,E1 -14640.285,E2 -14640.285} C_VEL
LIN {X 0,Y 332.079,Z 379.178,A -85,B 0,C 180,E1 -14642.732,E2 -14642.732} C_VEL
LIN {X 0,Y 332.515,Z 375.11,A -85,B 0,C 180,E1 -14644.993,E2 -14644.993} C_VEL
LIN {X 0,Y 333.004,Z 370.045,A -85,B 0,C 180,E1 -14647.018,E2 -14647.018} C_VEL
LIN {X 0,Y 333.674,Z 363.479,A -85,B 0,C 180,E1 -14649.019,E2 -14649.019} C_VEL
LIN {X 0,Y 334.641,Z 355.559,A -85,B 0,C 180,E1 -14650.923,E2 -14650.923} C_VEL
LIN {X 0,Y 335.747,Z 346.532,A -85,B 0,C 180,E1 -14652.645,E2 -14652.645} C_VEL
LIN {X 0,Y 336.934,Z 335.902,A -85,B 0,C 180,E1 -14654.266,E2 -14654.266} C_VEL
LIN {X 0,Y 338.137,Z 325.24,A -85,B 0,C 180,E1 -14655.557,E2 -14655.557} C_VEL
LIN {X 0,Y 339.13,Z 313.43,A -85,B 0,C 180,E1 -14656.686,E2 -14656.686} C_VEL
LIN {X 0,Y 340.072,Z 300.615,A -85,B 0,C 180,E1 -14657.619,E2 -14657.619} C_VEL
LIN {X 0,Y 340.886,Z 287.354,A -85,B 0,C 180,E1 -14658.291,E2 -14658.291} C_VEL
LIN {X 0,Y 341.425,Z 273.789,A -85,B 0,C 180,E1 -14658.723,E2 -14658.723} C_VEL
LIN {X 0,Y 342.907,Z 200.266,A -85,B 0,C 180,E1 -14660.332,E2 -14660.332} C_VEL
LIN {X 0,Y 339.277,Z 181.909,A -85,B 0,C 180,E1 -14660.987,E2 -14660.987} C_VEL
LIN {X 0,Y 335.803,Z 171.8,A -85,B 0,C 180,E1 -14661.462,E2 -14661.462} C_VEL
LIN {X 0,Y 333.907,Z 161.895,A -85,B 0,C 180,E1 -14664.489,E2 -14664.489} C_VEL
LIN {X 0,Y 334.102,Z 161.865,A -85,B 0,C 180,E1 -14667.589,E2 -14667.589} C_VEL
LIN {X 0,Y 334.08,Z 161.868,A -85,B 0,C 180,E1 -14671.205,E2 -14671.205} C_VEL
LIN {X 0,Y 333.807,Z 161.902,A -85,B 0,C 180,E1 -14673.621,E2 -14673.621} C_VEL
LIN {X 0,Y 333.991,Z 161.883,A -85,B 0,C 180,E1 -14676.039,E2 -14676.039} C_VEL
LIN {X 0,Y 333.851,Z 161.898,A -85,B 0,C 180,E1 -14679.695,E2 -14679.695} C_VEL
LIN {X 0,Y 333.789,Z 161.904,A -85,B 0,C 180,E1 -14683.392,E2 -14683.392} C_VEL
LIN {X 0,Y 333.702,Z 161.914,A -85,B 0,C 180,E1 -14687.149,E2 -14687.149} C_VEL
LIN {X 0,Y 333.687,Z 161.92,A -85,B 0,C 180,E1 -14689.694,E2 -14689.694} C_VEL
LIN {X 0,Y 333.644,Z 161.925,A -85,B 0,C 180,E1 -14693.592,E2 -14693.592} C_VEL
LIN {X 0,Y 333.669,Z 161.923,A -85,B 0,C 180,E1 -14697.606,E2 -14697.606} C_VEL
LIN {X 0,Y 333.618,Z 161.924,A -85,B 0,C 180,E1 -14701.309,E2 -14701.309} C_VEL
LIN {X 0,Y 332.955,Z 162.01,A -85,B 0,C 180,E1 -14702.317,E2 -14702.317} C_VEL
LIN {X 0,Y 330.09,Z 162.366,A -85,B 0,C 180,E1 -14703.957,E2 -14703.957} C_VEL
LIN {X 0,Y 327.678,Z 162.667,A -85,B 0,C 180,E1 -14705.285,E2 -14705.285} C_VEL
LIN {X 0,Y 326.67,Z 162.79,A -85,B 0,C 180,E1 -14706.313,E2 -14706.313} C_VEL
LIN {X 0,Y 326.603,Z 162.798,A -85,B 0,C 180,E1 -14706.661,E2 -14706.661} C_VEL
LIN {X 0,Y 326.558,Z 162.805,A -85,B 0,C 180,E1 -14710.214,E2 -14710.214} C_VEL
LIN {X 0,Y 326.562,Z 162.806,A -85,B 0,C 180,E1 -14713.526,E2 -14713.526} C_VEL
LIN {X 0,Y 326.575,Z 162.802,A -85,B 0,C 180,E1 -14717.029,E2 -14717.029} C_VEL
LIN {X 0,Y 326.584,Z 162.804,A -85,B 0,C 180,E1 -14721.386,E2 -14721.386} C_VEL
LIN {X 0,Y 326.621,Z 162.801,A -85,B 0,C 180,E1 -14724.852,E2 -14724.852} C_VEL
LIN {X 0,Y 326.61,Z 162.798,A -85,B 0,C 180,E1 -14727.456,E2 -14727.456} C_VEL
LIN {X 0,Y 326.618,Z 162.798,A -85,B 0,C 180,E1 -14730.337,E2 -14730.337} C_VEL
LIN {X 0,Y 326.644,Z 162.798,A -85,B 0,C 180,E1 -14734.645,E2 -14734.645} C_VEL
LIN {X 0,Y 326.613,Z 162.801,A -85,B 0,C 180,E1 -14738.543,E2 -14738.543} C_VEL
LIN {X 0,Y 326.651,Z 162.794,A -85,B 0,C 180,E1 -14741.206,E2 -14741.206} C_VEL
LIN {X 0,Y 326.728,Z 162.782,A -85,B 0,C 180,E1 -14745.459,E2 -14745.459} C_VEL
LIN {X 0,Y 326.761,Z 162.781,A -85,B 0,C 180,E1 -14748.839,E2 -14748.839} C_VEL
LIN {X 0,Y 326.917,Z 162.763,A -85,B 0,C 180,E1 -14752.589,E2 -14752.589} C_VEL
LIN {X 0,Y 326.75,Z 162.78,A -85,B 0,C 180,E1 -14755.064,E2 -14755.064} C_VEL
LIN {X 0,Y 327.012,Z 162.748,A -85,B 0,C 180,E1 -14757.536,E2 -14757.536} C_VEL
LIN {X 0,Y 327.032,Z 162.745,A -85,B 0,C 180,E1 -14761.231,E2 -14761.231} C_VEL
LIN {X 0,Y 326.751,Z 162.781,A -85,B 0,C 180,E1 -14763.7,E2 -14763.7} C_VEL
LIN {X 0,Y 326.946,Z 162.757,A -85,B 0,C 180,E1 -14766.17,E2 -14766.17} C_VEL
LIN {X 0,Y 326.783,Z 162.78,A -85,B 0,C 180,E1 -14769.907,E2 -14769.907} C_VEL
LIN {X 0,Y 326.725,Z 162.788,A -85,B 0,C 180,E1 -14773.687,E2 -14773.687} C_VEL
LIN {X 0,Y 326.623,Z 162.799,A -85,B 0,C 180,E1 -14777.532,E2 -14777.532} C_VEL
LIN {X 0,Y 326.604,Z 162.8,A -85,B 0,C 180,E1 -14781.458,E2 -14781.458} C_VEL
LIN {X 0,Y 326.601,Z 162.804,A -85,B 0,C 180,E1 -14785.491,E2 -14785.491} C_VEL
LIN {X 0,Y 326.591,Z 162.8,A -85,B 0,C 180,E1 -14788.257,E2 -14788.257} C_VEL
LIN {X 0,Y 326.575,Z 162.805,A -85,B 0,C 180,E1 -14791.097,E2 -14791.097} C_VEL
LIN {X 0,Y 326.608,Z 162.799,A -85,B 0,C 180,E1 -14794.019,E2 -14794.019} C_VEL
LIN {X 0,Y 326.623,Z 162.802,A -85,B 0,C 180,E1 -14797.237,E2 -14797.237} C_VEL
LIN {X 0,Y 326.545,Z 162.811,A -85,B 0,C 180,E1 -14801.124,E2 -14801.124} C_VEL
LIN {X 0,Y 326.56,Z 162.806,A -85,B 0,C 180,E1 -14803.526,E2 -14803.526} C_VEL
LIN {X 0,Y 326.573,Z 162.808,A -85,B 0,C 180,E1 -14807.029,E2 -14807.029} C_VEL
LIN {X 0,Y 326.583,Z 162.803,A -85,B 0,C 180,E1 -14811.385,E2 -14811.385} C_VEL
LIN {X 0,Y 326.619,Z 162.802,A -85,B 0,C 180,E1 -14814.852,E2 -14814.852} C_VEL
LIN {X 0,Y 326.646,Z 162.826,A -85,B 0,C 180,E1 -14818.946,E2 -14818.946} C_VEL
LIN {X 0,Y 328.995,Z 174.447,A -85,B 0,C 180,E1 -14822.314,E2 -14822.314} C_VEL
LIN {X 0,Y 330.606,Z 183.516,A -85,B 0,C 180,E1 -14824.839,E2 -14824.839} C_VEL
LIN {X 0,Y 330.073,Z 188.746,A -85,B 0,C 180,E1 -14826.178,E2 -14826.178} C_VEL
LIN {X 0,Y 335.248,Z 222.199,A -85,B 0,C 180,E1 -14827.335,E2 -14827.335} C_VEL
LIN {X 0,Y 335.86,Z 228.02,A -85,B 0,C 180,E1 -14827.511,E2 -14827.511} C_VEL
LIN {X 0,Y 334.232,Z 297.785,A -85,B 0,C 180,E1 -14829.096,E2 -14829.096} C_VEL
LIN {X 0,Y 333.537,Z 311.375,A -85,B 0,C 180,E1 -14829.655,E2 -14829.655} C_VEL
LIN {X 0,Y 332.558,Z 323.702,A -85,B 0,C 180,E1 -14830.398,E2 -14830.398} C_VEL
LIN {X 0,Y 331.313,Z 336.364,A -85,B 0,C 180,E1 -14831.446,E2 -14831.446} C_VEL
LIN {X 0,Y 330.067,Z 347.661,A -85,B 0,C 180,E1 -14832.657,E2 -14832.657} C_VEL
LIN {X 0,Y 328.894,Z 358.07,A -85,B 0,C 180,E1 -14834.068,E2 -14834.068} C_VEL
LIN {X 0,Y 327.735,Z 367.842,A -85,B 0,C 180,E1 -14835.723,E2 -14835.723} C_VEL
LIN {X 0,Y 326.672,Z 376.637,A -85,B 0,C 180,E1 -14837.576,E2 -14837.576} C_VEL
LIN {X 0,Y 325.89,Z 383.636,A -85,B 0,C 180,E1 -14839.437,E2 -14839.437} C_VEL
LIN {X 0,Y 325.369,Z 389.234,A -85,B 0,C 180,E1 -14841.303,E2 -14841.303} C_VEL
LIN {X 0,Y 325.054,Z 393.612,A -85,B 0,C 180,E1 -14843.17,E2 -14843.17} C_VEL
LIN {X 0,Y 324.892,Z 396.894,A -85,B 0,C 180,E1 -14845.036,E2 -14845.036} C_VEL
LIN {X 0,Y 324.899,Z 398.521,A -85,B 0,C 180,E1 -14846.279,E2 -14846.279} C_VEL
LIN {X 0,Y 324.837,Z 399.735,A -85,B 0,C 180,E1 -14847.52,E2 -14847.52} C_VEL
LIN {X 0,Y 324.833,Z 400.502,A -85,B 0,C 180,E1 -14848.76,E2 -14848.76} C_VEL
LIN {X 0,Y 324.874,Z 400.859,A -85,B 0,C 180,E1 -14850,E2 -14850} C_VEL
LIN {X 0,Y 324.834,Z 400.395,A -85,B 0,C 180,E1 -14852.48,E2 -14852.48} C_VEL
LIN {X 0,Y 324.874,Z 399.535,A -85,B 0,C 180,E1 -14853.721,E2 -14853.721} C_VEL
LIN {X 0,Y 324.909,Z 397.289,A -85,B 0,C 180,E1 -14855.723,E2 -14855.723} C_VEL
LIN {X 0,Y 325.285,Z 393.208,A -85,B 0,C 180,E1 -14858.073,E2 -14858.073} C_VEL
LIN {X 0,Y 325.786,Z 388.768,A -85,B 0,C 180,E1 -14859.938,E2 -14859.938} C_VEL
LIN {X 0,Y 326.501,Z 383.135,A -85,B 0,C 180,E1 -14861.8,E2 -14861.8} C_VEL
LIN {X 0,Y 327.638,Z 376.118,A -85,B 0,C 180,E1 -14863.648,E2 -14863.648} C_VEL
LIN {X 0,Y 328.999,Z 367.343,A -85,B 0,C 180,E1 -14865.487,E2 -14865.487} C_VEL
LIN {X 0,Y 330.255,Z 358.382,A -85,B 0,C 180,E1 -14867.014,E2 -14867.014} C_VEL
LIN {X 0,Y 331.868,Z 347.351,A -85,B 0,C 180,E1 -14868.521,E2 -14868.521} C_VEL
LIN {X 0,Y 333.347,Z 336.23,A -85,B 0,C 180,E1 -14869.715,E2 -14869.715} C_VEL
LIN {X 0,Y 334.861,Z 323.81,A -85,B 0,C 180,E1 -14870.743,E2 -14870.743} C_VEL
LIN {X 0,Y 335.965,Z 311.267,A -85,B 0,C 180,E1 -14871.515,E2 -14871.515} C_VEL
LIN {X 0,Y 336.894,Z 298.157,A -85,B 0,C 180,E1 -14872.056,E2 -14872.056} C_VEL
LIN {X 0,Y 337.66,Z 269.884,A -85,B 0,C 180,E1 -14872.74,E2 -14872.74} C_VEL
LIN {X 0,Y 338.72,Z 226.837,A -85,B 0,C 180,E1 -14873.718,E2 -14873.718} C_VEL
LIN {X 0,Y 335.177,Z 204.752,A -85,B 0,C 180,E1 -14874.581,E2 -14874.581} C_VEL
LIN {X 0,Y 331.594,Z 187.626,A -85,B 0,C 180,E1 -14875.375,E2 -14875.375} C_VEL
LIN {X 0,Y 331.241,Z 183.72,A -85,B 0,C 180,E1 -14876.46,E2 -14876.46} C_VEL
LIN {X 0,Y 328.945,Z 172.514,A -85,B 0,C 180,E1 -14879.785,E2 -14879.785} C_VEL
LIN {X 0,Y 326.605,Z 162.809,A -85,B 0,C 180,E1 -14882.896,E2 -14882.896} C_VEL
LIN {X 0,Y 326.611,Z 162.803,A -85,B 0,C 180,E1 -14885.52,E2 -14885.52} C_VEL
LIN {X 0,Y 326.589,Z 162.806,A -85,B 0,C 180,E1 -14889.222,E2 -14889.222} C_VEL
LIN {X 0,Y 326.573,Z 162.81,A -85,B 0,C 180,E1 -14892.971,E2 -14892.971} C_VEL
LIN {X 0,Y 326.573,Z 162.804,A -85,B 0,C 180,E1 -14897.029,E2 -14897.029} C_VEL
LIN {X 0,Y 326.583,Z 162.805,A -85,B 0,C 180,E1 -14901.386,E2 -14901.386} C_VEL
LIN {X 0,Y 326.62,Z 162.801,A -85,B 0,C 180,E1 -14904.852,E2 -14904.852} C_VEL
LIN {X 0,Y 326.61,Z 162.795,A -85,B 0,C 180,E1 -14907.456,E2 -14907.456} C_VEL
LIN {X 0,Y 326.581,Z 162.798,A -85,B 0,C 180,E1 -14910.333,E2 -14910.333} C_VEL
LIN {X 0,Y 326.597,Z 162.801,A -85,B 0,C 180,E1 -14913.135,E2 -14913.135} C_VEL
LIN {X 0,Y 326.593,Z 162.802,A -85,B 0,C 180,E1 -14917.211,E2 -14917.211} C_VEL
LIN {X 0,Y 326.632,Z 162.797,A -85,B 0,C 180,E1 -14921.216,E2 -14921.216} C_VEL
LIN {X 0,Y 326.718,Z 162.783,A -85,B 0,C 180,E1 -14925.467,E2 -14925.467} C_VEL
LIN {X 0,Y 326.752,Z 162.771,A -85,B 0,C 180,E1 -14928.838,E2 -14928.838} C_VEL
LIN {X 0,Y 326.929,Z 162.751,A -85,B 0,C 180,E1 -14932.589,E2 -14932.589} C_VEL
LIN {X 0,Y 326.747,Z 162.78,A -85,B 0,C 180,E1 -14935.064,E2 -14935.064} C_VEL
LIN {X 0,Y 327.005,Z 162.741,A -85,B 0,C 180,E1 -14937.536,E2 -14937.536} C_VEL
LIN {X 0,Y 327.031,Z 162.743,A -85,B 0,C 180,E1 -14941.231,E2 -14941.231} C_VEL
LIN {X 0,Y 326.741,Z 162.784,A -85,B 0,C 180,E1 -14943.7,E2 -14943.7} C_VEL
LIN {X 0,Y 326.923,Z 162.756,A -85,B 0,C 180,E1 -14946.459,E2 -14946.459} C_VEL
LIN {X 0,Y 326.785,Z 162.775,A -85,B 0,C 180,E1 -14949.907,E2 -14949.907} C_VEL
LIN {X 0,Y 326.746,Z 162.784,A -85,B 0,C 180,E1 -14953.686,E2 -14953.686} C_VEL
LIN {X 0,Y 326.63,Z 162.799,A -85,B 0,C 180,E1 -14957.532,E2 -14957.532} C_VEL
LIN {X 0,Y 326.605,Z 162.803,A -85,B 0,C 180,E1 -14961.458,E2 -14961.458} C_VEL
LIN {X 0,Y 326.603,Z 162.807,A -85,B 0,C 180,E1 -14965.491,E2 -14965.491} C_VEL
LIN {X 0,Y 326.643,Z 162.902,A -85,B 0,C 180,E1 -14969.219,E2 -14969.219} C_VEL
LIN {X 0,Y 328.924,Z 172.655,A -85,B 0,C 180,E1 -14972.423,E2 -14972.423} C_VEL
LIN {X 0,Y 335.757,Z 188.464,A -85,B 0,C 180,E1 -14973.502,E2 -14973.502} C_VEL
LIN {X 0,Y 337.45,Z 193.327,A -85,B 0,C 180,E1 -14973.777,E2 -14973.777} C_VEL
LIN {X 0,Y 339.427,Z 202.984,A -85,B 0,C 180,E1 -14974.192,E2 -14974.192} C_VEL
LIN {X 0,Y 337.223,Z 280.905,A -85,B 0,C 180,E1 -14975.981,E2 -14975.981} C_VEL
LIN {X 0,Y 336.371,Z 294.506,A -85,B 0,C 180,E1 -14976.541,E2 -14976.541} C_VEL
LIN {X 0,Y 335.443,Z 307.371,A -85,B 0,C 180,E1 -14977.348,E2 -14977.348} C_VEL
LIN {X 0,Y 334.087,Z 319.911,A -85,B 0,C 180,E1 -14978.407,E2 -14978.407} C_VEL
LIN {X 0,Y 332.686,Z 330.778,A -85,B 0,C 180,E1 -14979.588,E2 -14979.588} C_VEL
LIN {X 0,Y 331.214,Z 341.231,A -85,B 0,C 180,E1 -14981.029,E2 -14981.029} C_VEL
LIN {X 0,Y 329.875,Z 350.008,A -85,B 0,C 180,E1 -14982.523,E2 -14982.523} C_VEL
LIN {X 0,Y 328.593,Z 358.193,A -85,B 0,C 180,E1 -14984.234,E2 -14984.234} C_VEL
LIN {X 0,Y 327.372,Z 365.658,A -85,B 0,C 180,E1 -14986.184,E2 -14986.184} C_VEL
LIN {X 0,Y 326.451,Z 371.491,A -85,B 0,C 180,E1 -14988.134,E2 -14988.134} C_VEL
LIN {X 0,Y 325.696,Z 376.626,A -85,B 0,C 180,E1 -14990.398,E2 -14990.398} C_VEL
LIN {X 0,Y 325.102,Z 380.308,A -85,B 0,C 180,E1 -14992.749,E2 -14992.749} C_VEL
LIN {X 0,Y 324.845,Z 381.853,A -85,B 0,C 180,E1 -14994.257,E2 -14994.257} C_VEL
LIN {X 0,Y 324.685,Z 382.791,A -85,B 0,C 180,E1 -14995.751,E2 -14995.751} C_VEL
LIN {X 0,Y 324.576,Z 383.159,A -85,B 0,C 180,E1 -14997.615,E2 -14997.615} C_VEL
LIN {X 0,Y 324.659,Z 382.289,A -85,B 0,C 180,E1 -14999.985,E2 -14999.985} C_VEL
LIN {X 0,Y 324.94,Z 379.822,A -85,B 0,C 180,E1 -15002.471,E2 -15002.471} C_VEL
LIN {X 0,Y 325.262,Z 376.71,A -85,B 0,C 180,E1 -15004.396,E2 -15004.396} C_VEL
LIN {X 0,Y 325.75,Z 372.051,A -85,B 0,C 180,E1 -15006.476,E2 -15006.476} C_VEL
LIN {X 0,Y 326.423,Z 365.999,A -85,B 0,C 180,E1 -15008.53,E2 -15008.53} C_VEL
LIN {X 0,Y 327.247,Z 359.023,A -85,B 0,C 180,E1 -15010.397,E2 -15010.397} C_VEL
LIN {X 0,Y 328.389,Z 350.314,A -85,B 0,C 180,E1 -15012.243,E2 -15012.243} C_VEL
LIN {X 0,Y 329.507,Z 340.582,A -85,B 0,C 180,E1 -15013.902,E2 -15013.902} C_VEL
LIN {X 0,Y 330.634,Z 330.988,A -85,B 0,C 180,E1 -15015.222,E2 -15015.222} C_VEL
LIN {X 0,Y 331.718,Z 320.698,A -85,B 0,C 180,E1 -15016.367,E2 -15016.367} C_VEL
LIN {X 0,Y 332.714,Z 309.159,A -85,B 0,C 180,E1 -15017.38,E2 -15017.38} C_VEL
LIN {X 0,Y 333.564,Z 296.49,A -85,B 0,C 180,E1 -15018.222,E2 -15018.222} C_VEL
LIN {X 0,Y 334.308,Z 283.781,A -85,B 0,C 180,E1 -15018.806,E2 -15018.806} C_VEL
LIN {X 0,Y 334.782,Z 267.844,A -85,B 0,C 180,E1 -15019.236,E2 -15019.236} C_VEL
LIN {X 0,Y 336.239,Z 201.422,A -85,B 0,C 180,E1 -15020.716,E2 -15020.716} C_VEL
LIN {X 0,Y 332.81,Z 184.053,A -85,B 0,C 180,E1 -15021.352,E2 -15021.352} C_VEL
LIN {X 0,Y 328.664,Z 171.996,A -85,B 0,C 180,E1 -15021.933,E2 -15021.933} C_VEL
LIN {X 0,Y 326.802,Z 162.779,A -85,B 0,C 180,E1 -15024.795,E2 -15024.795} C_VEL
LIN {X 0,Y 327.043,Z 162.745,A -85,B 0,C 180,E1 -15027.537,E2 -15027.537} C_VEL
LIN {X 0,Y 327.048,Z 162.744,A -85,B 0,C 180,E1 -15031.231,E2 -15031.231} C_VEL
LIN {X 0,Y 326.756,Z 162.781,A -85,B 0,C 180,E1 -15033.7,E2 -15033.7} C_VEL
LIN {X 0,Y 326.945,Z 162.762,A -85,B 0,C 180,E1 -15036.17,E2 -15036.17} C_VEL
LIN {X 0,Y 326.806,Z 162.777,A -85,B 0,C 180,E1 -15039.907,E2 -15039.907} C_VEL
LIN {X 0,Y 326.745,Z 162.784,A -85,B 0,C 180,E1 -15043.686,E2 -15043.686} C_VEL
LIN {X 0,Y 326.653,Z 162.793,A -85,B 0,C 180,E1 -15047.531,E2 -15047.531} C_VEL
LIN {X 0,Y 326.63,Z 162.799,A -85,B 0,C 180,E1 -15050.137,E2 -15050.137} C_VEL
LIN {X 0,Y 326.593,Z 162.799,A -85,B 0,C 180,E1 -15052.79,E2 -15052.79} C_VEL
LIN {X 0,Y 326.604,Z 162.799,A -85,B 0,C 180,E1 -15056.865,E2 -15056.865} C_VEL
LIN {X 0,Y 326.613,Z 162.797,A -85,B 0,C 180,E1 -15060.603,E2 -15060.603} C_VEL
LIN {X 0,Y 326.609,Z 162.798,A -85,B 0,C 180,E1 -15064.019,E2 -15064.019} C_VEL
LIN {X 0,Y 326.603,Z 162.798,A -85,B 0,C 180,E1 -15066.661,E2 -15066.661} C_VEL
LIN {X 0,Y 325.964,Z 162.882,A -85,B 0,C 180,E1 -15067.69,E2 -15067.69} C_VEL
LIN {X 0,Y 323.082,Z 163.243,A -85,B 0,C 180,E1 -15069.362,E2 -15069.362} C_VEL
LIN {X 0,Y 320.624,Z 163.547,A -85,B 0,C 180,E1 -15070.717,E2 -15070.717} C_VEL
LIN {X 0,Y 319.58,Z 163.676,A -85,B 0,C 180,E1 -15071.767,E2 -15071.767} C_VEL
LIN {X 0,Y 319.502,Z 163.683,A -85,B 0,C 180,E1 -15072.123,E2 -15072.123} C_VEL
LIN {X 0,Y 319.489,Z 163.686,A -85,B 0,C 180,E1 -15075.257,E2 -15075.257} C_VEL
LIN {X 0,Y 319.507,Z 163.68,A -85,B 0,C 180,E1 -15078.407,E2 -15078.407} C_VEL
LIN {X 0,Y 319.534,Z 163.679,A -85,B 0,C 180,E1 -15081.986,E2 -15081.986} C_VEL
LIN {X 0,Y 319.562,Z 163.68,A -85,B 0,C 180,E1 -15085.123,E2 -15085.123} C_VEL
LIN {X 0,Y 319.527,Z 163.679,A -85,B 0,C 180,E1 -15088.137,E2 -15088.137} C_VEL
LIN {X 0,Y 319.573,Z 163.675,A -85,B 0,C 180,E1 -15091.604,E2 -15091.604} C_VEL
LIN {X 0,Y 319.575,Z 163.675,A -85,B 0,C 180,E1 -15095.301,E2 -15095.301} C_VEL
LIN {X 0,Y 319.566,Z 163.675,A -85,B 0,C 180,E1 -15098.045,E2 -15098.045} C_VEL
LIN {X 0,Y 319.59,Z 163.674,A -85,B 0,C 180,E1 -15102.069,E2 -15102.069} C_VEL
LIN {X 0,Y 319.713,Z 163.657,A -85,B 0,C 180,E1 -15106.007,E2 -15106.007} C_VEL
LIN {X 0,Y 319.739,Z 163.655,A -85,B 0,C 180,E1 -15109.872,E2 -15109.872} C_VEL
LIN {X 0,Y 319.903,Z 163.633,A -85,B 0,C 180,E1 -15113.693,E2 -15113.693} C_VEL
LIN {X 0,Y 319.958,Z 163.627,A -85,B 0,C 180,E1 -15117.482,E2 -15117.482} C_VEL
LIN {X 0,Y 320.001,Z 163.621,A -85,B 0,C 180,E1 -15121.258,E2 -15121.258} C_VEL
LIN {X 0,Y 319.701,Z 163.659,A -85,B 0,C 180,E1 -15123.781,E2 -15123.781} C_VEL
LIN {X 0,Y 319.903,Z 163.631,A -85,B 0,C 180,E1 -15126.306,E2 -15126.306} C_VEL
LIN {X 0,Y 319.735,Z 163.657,A -85,B 0,C 180,E1 -15130.128,E2 -15130.128} C_VEL
LIN {X 0,Y 319.696,Z 163.663,A -85,B 0,C 180,E1 -15133.994,E2 -15133.994} C_VEL
LIN {X 0,Y 319.576,Z 163.676,A -85,B 0,C 180,E1 -15137.932,E2 -15137.932} C_VEL
LIN {X 0,Y 319.562,Z 163.677,A -85,B 0,C 180,E1 -15141.955,E2 -15141.955} C_VEL
LIN {X 0,Y 319.55,Z 163.679,A -85,B 0,C 180,E1 -15146.095,E2 -15146.095} C_VEL
LIN {X 0,Y 319.526,Z 163.681,A -85,B 0,C 180,E1 -15148.94,E2 -15148.94} C_VEL
LIN {X 0,Y 319.526,Z 163.682,A -85,B 0,C 180,E1 -15151.863,E2 -15151.863} C_VEL
LIN {X 0,Y 319.58,Z 163.678,A -85,B 0,C 180,E1 -15155.542,E2 -15155.542} C_VEL
LIN {X 0,Y 319.53,Z 163.682,A -85,B 0,C 180,E1 -15159.662,E2 -15159.662} C_VEL
LIN {X 0,Y 319.52,Z 163.684,A -85,B 0,C 180,E1 -15163.46,E2 -15163.46} C_VEL
LIN {X 0,Y 319.551,Z 163.682,A -85,B 0,C 180,E1 -15167.016,E2 -15167.016} C_VEL
LIN {X 0,Y 319.546,Z 163.679,A -85,B 0,C 180,E1 -15170.37,E2 -15170.37} C_VEL
LIN {X 0,Y 319.579,Z 163.677,A -85,B 0,C 180,E1 -15174.457,E2 -15174.457} C_VEL
LIN {X 0,Y 319.576,Z 163.679,A -85,B 0,C 180,E1 -15178.518,E2 -15178.518} C_VEL
LIN {X 0,Y 321.447,Z 172.645,A -85,B 0,C 180,E1 -15181.249,E2 -15181.249} C_VEL
LIN {X 0,Y 323.628,Z 184.341,A -85,B 0,C 180,E1 -15184.602,E2 -15184.602} C_VEL
LIN {X 0,Y 323.277,Z 188.643,A -85,B 0,C 180,E1 -15185.733,E2 -15185.733} C_VEL
LIN {X 0,Y 329.132,Z 227.036,A -85,B 0,C 180,E1 -15187.071,E2 -15187.071} C_VEL
LIN {X 0,Y 327.497,Z 296.893,A -85,B 0,C 180,E1 -15188.686,E2 -15188.686} C_VEL
LIN {X 0,Y 326.834,Z 309.95,A -85,B 0,C 180,E1 -15189.218,E2 -15189.218} C_VEL
LIN {X 0,Y 325.836,Z 322.615,A -85,B 0,C 180,E1 -15189.976,E2 -15189.976} C_VEL
LIN {X 0,Y 324.685,Z 333.928,A -85,B 0,C 180,E1 -15190.889,E2 -15190.889} C_VEL
LIN {X 0,Y 323.38,Z 345.635,A -85,B 0,C 180,E1 -15192.123,E2 -15192.123} C_VEL
LIN {X 0,Y 322.146,Z 356.179,A -85,B 0,C 180,E1 -15193.524,E2 -15193.524} C_VEL
LIN {X 0,Y 321.062,Z 365.673,A -85,B 0,C 180,E1 -15195.096,E2 -15195.096} C_VEL
LIN {X 0,Y 319.867,Z 374.811,A -85,B 0,C 180,E1 -15196.985,E2 -15196.985} C_VEL
LIN {X 0,Y 318.961,Z 382.169,A -85,B 0,C 180,E1 -15198.884,E2 -15198.884} C_VEL
LIN {X 0,Y 318.478,Z 387.139,A -85,B 0,C 180,E1 -15200.473,E2 -15200.473} C_VEL
LIN {X 0,Y 318.067,Z 391.952,A -85,B 0,C 180,E1 -15202.382,E2 -15202.382} C_VEL
LIN {X 0,Y 317.838,Z 395.623,A -85,B 0,C 180,E1 -15204.29,E2 -15204.29} C_VEL
LIN {X 0,Y 317.806,Z 398.256,A -85,B 0,C 180,E1 -15206.196,E2 -15206.196} C_VEL
LIN {X 0,Y 317.759,Z 399.487,A -85,B 0,C 180,E1 -15207.465,E2 -15207.465} C_VEL
LIN {X 0,Y 317.744,Z 400.284,A -85,B 0,C 180,E1 -15208.733,E2 -15208.733} C_VEL
LIN {X 0,Y 317.781,Z 400.656,A -85,B 0,C 180,E1 -15210,E2 -15210} C_VEL
LIN {X 0,Y 317.754,Z 400.221,A -85,B 0,C 180,E1 -15212.535,E2 -15212.535} C_VEL
LIN {X 0,Y 317.783,Z 399.39,A -85,B 0,C 180,E1 -15213.804,E2 -15213.804} C_VEL
LIN {X 0,Y 317.825,Z 397.402,A -85,B 0,C 180,E1 -15215.686,E2 -15215.686} C_VEL
LIN {X 0,Y 318.085,Z 394.371,A -85,B 0,C 180,E1 -15217.618,E2 -15217.618} C_VEL
LIN {X 0,Y 318.572,Z 390.329,A -85,B 0,C 180,E1 -15219.524,E2 -15219.524} C_VEL
LIN {X 0,Y 319.405,Z 384.132,A -85,B 0,C 180,E1 -15221.744,E2 -15221.744} C_VEL
LIN {X 0,Y 320.531,Z 377.39,A -85,B 0,C 180,E1 -15223.633,E2 -15223.633} C_VEL
LIN {X 0,Y 321.943,Z 369.095,A -85,B 0,C 180,E1 -15225.502,E2 -15225.502} C_VEL
LIN {X 0,Y 323.179,Z 360.528,A -85,B 0,C 180,E1 -15227.072,E2 -15227.072} C_VEL
LIN {X 0,Y 324.78,Z 350.014,A -85,B 0,C 180,E1 -15228.613,E2 -15228.613} C_VEL
LIN {X 0,Y 326.298,Z 339.643,A -85,B 0,C 180,E1 -15229.83,E2 -15229.83} C_VEL
LIN {X 0,Y 327.784,Z 328.309,A -85,B 0,C 180,E1 -15230.883,E2 -15230.883} C_VEL
LIN {X 0,Y 329.004,Z 316.734,A -85,B 0,C 180,E1 -15231.705,E2 -15231.705} C_VEL
LIN {X 0,Y 330.097,Z 303.584,A -85,B 0,C 180,E1 -15232.369,E2 -15232.369} C_VEL
LIN {X 0,Y 330.749,Z 290.477,A -85,B 0,C 180,E1 -15232.793,E2 -15232.793} C_VEL
LIN {X 0,Y 332.303,Z 227.131,A -85,B 0,C 180,E1 -15234.266,E2 -15234.266} C_VEL
LIN {X 0,Y 329.073,Z 206.878,A -85,B 0,C 180,E1 -15235.087,E2 -15235.087} C_VEL
LIN {X 0,Y 325.265,Z 189.315,A -85,B 0,C 180,E1 -15235.922,E2 -15235.922} C_VEL
LIN {X 0,Y 324.713,Z 187.299,A -85,B 0,C 180,E1 -15236.077,E2 -15236.077} C_VEL
LIN {X 0,Y 322.592,Z 176.338,A -85,B 0,C 180,E1 -15239.373,E2 -15239.373} C_VEL
LIN {X 0,Y 320.285,Z 166.562,A -85,B 0,C 180,E1 -15242.521,E2 -15242.521} C_VEL
LIN {X 0,Y 319.573,Z 163.682,A -85,B 0,C 180,E1 -15243.542,E2 -15243.542} C_VEL
LIN {X 0,Y 319.556,Z 163.679,A -85,B 0,C 180,E1 -15246.428,E2 -15246.428} C_VEL
LIN {X 0,Y 319.529,Z 163.683,A -85,B 0,C 180,E1 -15249.662,E2 -15249.662} C_VEL
LIN {X 0,Y 319.52,Z 163.687,A -85,B 0,C 180,E1 -15253.46,E2 -15253.46} C_VEL
LIN {X 0,Y 319.552,Z 163.678,A -85,B 0,C 180,E1 -15257.016,E2 -15257.016} C_VEL
LIN {X 0,Y 319.547,Z 163.675,A -85,B 0,C 180,E1 -15260.371,E2 -15260.371} C_VEL
LIN {X 0,Y 319.58,Z 163.674,A -85,B 0,C 180,E1 -15264.458,E2 -15264.458} C_VEL
LIN {X 0,Y 319.526,Z 163.679,A -85,B 0,C 180,E1 -15268.137,E2 -15268.137} C_VEL
LIN {X 0,Y 319.545,Z 163.675,A -85,B 0,C 180,E1 -15271.613,E2 -15271.613} C_VEL
LIN {X 0,Y 319.526,Z 163.673,A -85,B 0,C 180,E1 -15275.298,E2 -15275.298} C_VEL
LIN {X 0,Y 319.562,Z 163.678,A -85,B 0,C 180,E1 -15278.045,E2 -15278.045} C_VEL
LIN {X 0,Y 319.578,Z 163.678,A -85,B 0,C 180,E1 -15282.068,E2 -15282.068} C_VEL
LIN {X 0,Y 319.696,Z 163.659,A -85,B 0,C 180,E1 -15286.006,E2 -15286.006} C_VEL
LIN {X 0,Y 319.735,Z 163.648,A -85,B 0,C 180,E1 -15289.872,E2 -15289.872} C_VEL
LIN {X 0,Y 319.889,Z 163.63,A -85,B 0,C 180,E1 -15292.425,E2 -15292.425} C_VEL
LIN {X 0,Y 319.717,Z 163.656,A -85,B 0,C 180,E1 -15294.956,E2 -15294.956} C_VEL
LIN {X 0,Y 319.951,Z 163.62,A -85,B 0,C 180,E1 -15297.482,E2 -15297.482} C_VEL
LIN {X 0,Y 320.001,Z 163.618,A -85,B 0,C 180,E1 -15301.259,E2 -15301.259} C_VEL
LIN {X 0,Y 319.692,Z 163.662,A -85,B 0,C 180,E1 -15303.782,E2 -15303.782} C_VEL
LIN {X 0,Y 319.889,Z 163.632,A -85,B 0,C 180,E1 -15306.44,E2 -15306.44} C_VEL
LIN {X 0,Y 319.737,Z 163.654,A -85,B 0,C 180,E1 -15310.128,E2 -15310.128} C_VEL
LIN {X 0,Y 319.712,Z 163.663,A -85,B 0,C 180,E1 -15313.993,E2 -15313.993} C_VEL
LIN {X 0,Y 319.581,Z 163.674,A -85,B 0,C 180,E1 -15317.932,E2 -15317.932} C_VEL
LIN {X 0,Y 319.563,Z 163.68,A -85,B 0,C 180,E1 -15321.955,E2 -15321.955} C_VEL
LIN {X 0,Y 319.552,Z 163.683,A -85,B 0,C 180,E1 -15326.095,E2 -15326.095} C_VEL
LIN {X 0,Y 319.591,Z 163.766,A -85,B 0,C 180,E1 -15328.599,E2 -15328.599} C_VEL
LIN {X 0,Y 321.862,Z 173.104,A -85,B 0,C 180,E1 -15331.742,E2 -15331.742} C_VEL
LIN {X 0,Y 329.435,Z 190.291,A -85,B 0,C 180,E1 -15332.957,E2 -15332.957} C_VEL
LIN {X 0,Y 331.387,Z 195.597,A -85,B 0,C 180,E1 -15333.282,E2 -15333.282} C_VEL
LIN {X 0,Y 333.016,Z 203.592,A -85,B 0,C 180,E1 -15333.641,E2 -15333.641} C_VEL
LIN {X 0,Y 330.806,Z 281.131,A -85,B 0,C 180,E1 -15335.463,E2 -15335.463} C_VEL
LIN {X 0,Y 329.932,Z 294.613,A -85,B 0,C 180,E1 -15336.028,E2 -15336.028} C_VEL
LIN {X 0,Y 329.104,Z 305.785,A -85,B 0,C 180,E1 -15336.723,E2 -15336.723} C_VEL
LIN {X 0,Y 327.834,Z 317.747,A -85,B 0,C 180,E1 -15337.703,E2 -15337.703} C_VEL
LIN {X 0,Y 326.247,Z 329.733,A -85,B 0,C 180,E1 -15338.985,E2 -15338.985} C_VEL
LIN {X 0,Y 324.906,Z 339.049,A -85,B 0,C 180,E1 -15340.237,E2 -15340.237} C_VEL
LIN {X 0,Y 323.533,Z 347.913,A -85,B 0,C 180,E1 -15341.693,E2 -15341.693} C_VEL
LIN {X 0,Y 322.057,Z 356.714,A -85,B 0,C 180,E1 -15343.482,E2 -15343.482} C_VEL
LIN {X 0,Y 320.707,Z 364.505,A -85,B 0,C 180,E1 -15345.472,E2 -15345.472} C_VEL
LIN {X 0,Y 319.669,Z 370.59,A -85,B 0,C 180,E1 -15347.439,E2 -15347.439} C_VEL
LIN {X 0,Y 318.875,Z 375.409,A -85,B 0,C 180,E1 -15349.444,E2 -15349.444} C_VEL
LIN {X 0,Y 318.244,Z 379.488,A -85,B 0,C 180,E1 -15351.804,E2 -15351.804} C_VEL
LIN {X 0,Y 317.9,Z 381.379,A -85,B 0,C 180,E1 -15353.351,E2 -15353.351} C_VEL
LIN {X 0,Y 317.666,Z 382.626,A -85,B 0,C 180,E1 -15354.944,E2 -15354.944} C_VEL
LIN {X 0,Y 317.49,Z 383.358,A -85,B 0,C 180,E1 -15357.265,E2 -15357.265} C_VEL
LIN {X 0,Y 317.529,Z 382.674,A -85,B 0,C 180,E1 -15359.679,E2 -15359.679} C_VEL
LIN {X 0,Y 317.794,Z 380.391,A -85,B 0,C 180,E1 -15362.203,E2 -15362.203} C_VEL
LIN {X 0,Y 318.088,Z 378.116,A -85,B 0,C 180,E1 -15363.775,E2 -15363.775} C_VEL
LIN {X 0,Y 318.554,Z 373.9,A -85,B 0,C 180,E1 -15365.911,E2 -15365.911} C_VEL
LIN {X 0,Y 319.111,Z 368.368,A -85,B 0,C 180,E1 -15368.012,E2 -15368.012} C_VEL
LIN {X 0,Y 319.991,Z 361.247,A -85,B 0,C 180,E1 -15370.092,E2 -15370.092} C_VEL
LIN {X 0,Y 321.015,Z 353.819,A -85,B 0,C 180,E1 -15371.821,E2 -15371.821} C_VEL
LIN {X 0,Y 322.244,Z 344.031,A -85,B 0,C 180,E1 -15373.663,E2 -15373.663} C_VEL
LIN {X 0,Y 323.471,Z 333.643,A -85,B 0,C 180,E1 -15375.209,E2 -15375.209} C_VEL
LIN {X 0,Y 324.734,Z 322.408,A -85,B 0,C 180,E1 -15376.54,E2 -15376.54} C_VEL
LIN {X 0,Y 325.797,Z 310.803,A -85,B 0,C 180,E1 -15377.621,E2 -15377.621} C_VEL
LIN {X 0,Y 326.733,Z 297.842,A -85,B 0,C 180,E1 -15378.523,E2 -15378.523} C_VEL
LIN {X 0,Y 327.541,Z 284.547,A -85,B 0,C 180,E1 -15379.167,E2 -15379.167} C_VEL
LIN {X 0,Y 328.019,Z 269.397,A -85,B 0,C 180,E1 -15379.596,E2 -15379.596} C_VEL
LIN {X 0,Y 329.579,Z 202.429,A -85,B 0,C 180,E1 -15381.117,E2 -15381.117} C_VEL
LIN {X 0,Y 326.405,Z 186.246,A -85,B 0,C 180,E1 -15381.725,E2 -15381.725} C_VEL
LIN {X 0,Y 321.515,Z 172.204,A -85,B 0,C 180,E1 -15382.424,E2 -15382.424} C_VEL
LIN {X 0,Y 319.742,Z 163.657,A -85,B 0,C 180,E1 -15385.153,E2 -15385.153} C_VEL
LIN {X 0,Y 319.986,Z 163.625,A -85,B 0,C 180,E1 -15387.482,E2 -15387.482} C_VEL
LIN {X 0,Y 320.015,Z 163.62,A -85,B 0,C 180,E1 -15391.258,E2 -15391.258} C_VEL
LIN {X 0,Y 319.722,Z 163.657,A -85,B 0,C 180,E1 -15395.044,E2 -15395.044} C_VEL
LIN {X 0,Y 319.855,Z 163.64,A -85,B 0,C 180,E1 -15397.576,E2 -15397.576} C_VEL
LIN {X 0,Y 319.724,Z 163.655,A -85,B 0,C 180,E1 -15401.41,E2 -15401.41} C_VEL
LIN {X 0,Y 319.667,Z 163.663,A -85,B 0,C 180,E1 -15404.679,E2 -15404.679} C_VEL
LIN {X 0,Y 319.618,Z 163.673,A -85,B 0,C 180,E1 -15407.929,E2 -15407.929} C_VEL
LIN {X 0,Y 319.585,Z 163.674,A -85,B 0,C 180,E1 -15410.601,E2 -15410.601} C_VEL
LIN {X 0,Y 319.534,Z 163.68,A -85,B 0,C 180,E1 -15413.322,E2 -15413.322} C_VEL
LIN {X 0,Y 319.554,Z 163.679,A -85,B 0,C 180,E1 -15416.095,E2 -15416.095} C_VEL
LIN {X 0,Y 319.544,Z 163.679,A -85,B 0,C 180,E1 -15418.938,E2 -15418.938} C_VEL
LIN {X 0,Y 319.526,Z 163.681,A -85,B 0,C 180,E1 -15421.863,E2 -15421.863} C_VEL
LIN {X 0,Y 319.582,Z 163.677,A -85,B 0,C 180,E1 -15425.543,E2 -15425.543} C_VEL
LIN {X 0,Y 319.53,Z 163.683,A -85,B 0,C 180,E1 -15429.662,E2 -15429.662} C_VEL
LIN {X 0,Y 319.502,Z 163.683,A -85,B 0,C 180,E1 -15432.123,E2 -15432.123} C_VEL
LIN {X 0,Y 318.859,Z 163.767,A -85,B 0,C 180,E1 -15433.175,E2 -15433.175} C_VEL
LIN {X 0,Y 316.028,Z 164.118,A -85,B 0,C 180,E1 -15434.889,E2 -15434.889} C_VEL
LIN {X 0,Y 313.607,Z 164.42,A -85,B 0,C 180,E1 -15436.278,E2 -15436.278} C_VEL
LIN {X 0,Y 312.554,Z 164.548,A -85,B 0,C 180,E1 -15437.353,E2 -15437.353} C_VEL
LIN {X 0,Y 312.462,Z 164.558,A -85,B 0,C 180,E1 -15437.717,E2 -15437.717} C_VEL
LIN {X 0,Y 312.486,Z 164.557,A -85,B 0,C 180,E1 -15441.923,E2 -15441.923} C_VEL
LIN {X 0,Y 312.532,Z 164.552,A -85,B 0,C 180,E1 -15444.22,E2 -15444.22} C_VEL
LIN {X 0,Y 312.504,Z 164.555,A -85,B 0,C 180,E1 -15447.334,E2 -15447.334} C_VEL
LIN {X 0,Y 312.509,Z 164.557,A -85,B 0,C 180,E1 -15451.292,E2 -15451.292} C_VEL
LIN {X 0,Y 312.549,Z 164.554,A -85,B 0,C 180,E1 -15454.708,E2 -15454.708} C_VEL
LIN {X 0,Y 312.52,Z 164.557,A -85,B 0,C 180,E1 -15458.911,E2 -15458.911} C_VEL
LIN {X 0,Y 312.554,Z 164.549,A -85,B 0,C 180,E1 -15461.651,E2 -15461.651} C_VEL
LIN {X 0,Y 312.655,Z 164.534,A -85,B 0,C 180,E1 -15465.684,E2 -15465.684} C_VEL
LIN {X 0,Y 312.688,Z 164.532,A -85,B 0,C 180,E1 -15469.641,E2 -15469.641} C_VEL
LIN {X 0,Y 312.8,Z 164.522,A -85,B 0,C 180,E1 -15472.252,E2 -15472.252} C_VEL
LIN {X 0,Y 312.691,Z 164.532,A -85,B 0,C 180,E1 -15474.842,E2 -15474.842} C_VEL
LIN {X 0,Y 312.97,Z 164.499,A -85,B 0,C 180,E1 -15478.713,E2 -15478.713} C_VEL
LIN {X 0,Y 312.97,Z 164.496,A -85,B 0,C 180,E1 -15481.287,E2 -15481.287} C_VEL
LIN {X 0,Y 312.689,Z 164.527,A -85,B 0,C 180,E1 -15485.158,E2 -15485.158} C_VEL
LIN {X 0,Y 312.802,Z 164.514,A -85,B 0,C 180,E1 -15487.747,E2 -15487.747} C_VEL
LIN {X 0,Y 312.654,Z 164.539,A -85,B 0,C 180,E1 -15491.672,E2 -15491.672} C_VEL
LIN {X 0,Y 312.606,Z 164.543,A -85,B 0,C 180,E1 -15494.82,E2 -15494.82} C_VEL
LIN {X 0,Y 312.535,Z 164.549,A -85,B 0,C 180,E1 -15499.184,E2 -15499.184} C_VEL
LIN {X 0,Y 312.516,Z 164.552,A -85,B 0,C 180,E1 -15502.775,E2 -15502.775} C_VEL
LIN {X 0,Y 312.484,Z 164.558,A -85,B 0,C 180,E1 -15506.732,E2 -15506.732} C_VEL
LIN {X 0,Y 312.47,Z 164.563,A -85,B 0,C 180,E1 -15509.658,E2 -15509.658} C_VEL
LIN {X 0,Y 312.521,Z 164.556,A -85,B 0,C 180,E1 -15513.689,E2 -15513.689} C_VEL
LIN {X 0,Y 312.515,Z 164.559,A -85,B 0,C 180,E1 -15517.387,E2 -15517.387} C_VEL
LIN {X 0,Y 312.442,Z 164.565,A -85,B 0,C 180,E1 -15520.717,E2 -15520.717} C_VEL
LIN {X 0,Y 312.451,Z 164.562,A -85,B 0,C 180,E1 -15524.21,E2 -15524.21} C_VEL
LIN {X 0,Y 312.455,Z 164.562,A -85,B 0,C 180,E1 -15527.925,E2 -15527.925} C_VEL
LIN {X 0,Y 312.484,Z 164.558,A -85,B 0,C 180,E1 -15531.923,E2 -15531.923} C_VEL
LIN {X 0,Y 312.531,Z 164.554,A -85,B 0,C 180,E1 -15534.22,E2 -15534.22} C_VEL
LIN {X 0,Y 312.526,Z 164.621,A -85,B 0,C 180,E1 -15538.207,E2 -15538.207} C_VEL
LIN {X 0,Y 314.633,Z 174.737,A -85,B 0,C 180,E1 -15541.298,E2 -15541.298} C_VEL
LIN {X 0,Y 316.612,Z 185.144,A -85,B 0,C 180,E1 -15544.351,E2 -15544.351} C_VEL
LIN {X 0,Y 316.482,Z 188.728,A -85,B 0,C 180,E1 -15545.262,E2 -15545.262} C_VEL
LIN {X 0,Y 322.108,Z 225.36,A -85,B 0,C 180,E1 -15546.574,E2 -15546.574} C_VEL
LIN {X 0,Y 322.438,Z 230.505,A -85,B 0,C 180,E1 -15546.725,E2 -15546.725} C_VEL
LIN {X 0,Y 320.764,Z 297.127,A -85,B 0,C 180,E1 -15548.301,E2 -15548.301} C_VEL
LIN {X 0,Y 320.044,Z 310.797,A -85,B 0,C 180,E1 -15548.883,E2 -15548.883} C_VEL
LIN {X 0,Y 318.946,Z 323.693,A -85,B 0,C 180,E1 -15549.693,E2 -15549.693} C_VEL
LIN {X 0,Y 317.635,Z 336.272,A -85,B 0,C 180,E1 -15550.784,E2 -15550.784} C_VEL
LIN {X 0,Y 316.271,Z 347.514,A -85,B 0,C 180,E1 -15552.042,E2 -15552.042} C_VEL
LIN {X 0,Y 315.115,Z 357.215,A -85,B 0,C 180,E1 -15553.408,E2 -15553.408} C_VEL
LIN {X 0,Y 313.924,Z 366.793,A -85,B 0,C 180,E1 -15555.081,E2 -15555.081} C_VEL
LIN {X 0,Y 312.725,Z 375.714,A -85,B 0,C 180,E1 -15557.013,E2 -15557.013} C_VEL
LIN {X 0,Y 311.867,Z 382.843,A -85,B 0,C 180,E1 -15558.957,E2 -15558.957} C_VEL
LIN {X 0,Y 311.272,Z 388.523,A -85,B 0,C 180,E1 -15560.906,E2 -15560.906} C_VEL
LIN {X 0,Y 310.918,Z 392.978,A -85,B 0,C 180,E1 -15562.858,E2 -15562.858} C_VEL
LIN {X 0,Y 310.712,Z 396.33,A -85,B 0,C 180,E1 -15564.809,E2 -15564.809} C_VEL
LIN {X 0,Y 310.717,Z 397.991,A -85,B 0,C 180,E1 -15566.109,E2 -15566.109} C_VEL
LIN {X 0,Y 310.682,Z 399.238,A -85,B 0,C 180,E1 -15567.407,E2 -15567.407} C_VEL
LIN {X 0,Y 310.658,Z 400.065,A -85,B 0,C 180,E1 -15568.704,E2 -15568.704} C_VEL
LIN {X 0,Y 310.691,Z 400.453,A -85,B 0,C 180,E1 -15570,E2 -15570} C_VEL
LIN {X 0,Y 310.677,Z 400.047,A -85,B 0,C 180,E1 -15572.593,E2 -15572.593} C_VEL
LIN {X 0,Y 310.695,Z 399.243,A -85,B 0,C 180,E1 -15573.891,E2 -15573.891} C_VEL
LIN {X 0,Y 310.822,Z 396.341,A -85,B 0,C 180,E1 -15576.492,E2 -15576.492} C_VEL
LIN {X 0,Y 311.19,Z 393.039,A -85,B 0,C 180,E1 -15578.442,E2 -15578.442} C_VEL
LIN {X 0,Y 311.746,Z 388.671,A -85,B 0,C 180,E1 -15580.39,E2 -15580.39} C_VEL
LIN {X 0,Y 312.757,Z 382.094,A -85,B 0,C 180,E1 -15582.656,E2 -15582.656} C_VEL
LIN {X 0,Y 314.09,Z 374.889,A -85,B 0,C 180,E1 -15584.58,E2 -15584.58} C_VEL
LIN {X 0,Y 315.383,Z 366.787,A -85,B 0,C 180,E1 -15586.337,E2 -15586.337} C_VEL
LIN {X 0,Y 317.05,Z 356.812,A -85,B 0,C 180,E1 -15588.08,E2 -15588.08} C_VEL
LIN {X 0,Y 318.637,Z 346.713,A -85,B 0,C 180,E1 -15589.488,E2 -15589.488} C_VEL
LIN {X 0,Y 320.269,Z 335.536,A -85,B 0,C 180,E1 -15590.723,E2 -15590.723} C_VEL
LIN {X 0,Y 321.946,Z 323.04,A -85,B 0,C 180,E1 -15591.784,E2 -15591.784} C_VEL
LIN {X 0,Y 323.038,Z 311.07,A -85,B 0,C 180,E1 -15592.548,E2 -15592.548} C_VEL
LIN {X 0,Y 324.066,Z 297.656,A -85,B 0,C 180,E1 -15593.121,E2 -15593.121} C_VEL
LIN {X 0,Y 324.962,Z 268.788,A -85,B 0,C 180,E1 -15593.846,E2 -15593.846} C_VEL
LIN {X 0,Y 326.053,Z 228.413,A -85,B 0,C 180,E1 -15594.805,E2 -15594.805} C_VEL
LIN {X 0,Y 322.807,Z 208.125,A -85,B 0,C 180,E1 -15595.66,E2 -15595.66} C_VEL
LIN {X 0,Y 319.348,Z 191.872,A -85,B 0,C 180,E1 -15596.451,E2 -15596.451} C_VEL
LIN {X 0,Y 317.553,Z 187.142,A -85,B 0,C 180,E1 -15596.798,E2 -15596.798} C_VEL
LIN {X 0,Y 315.383,Z 176.332,A -85,B 0,C 180,E1 -15600.173,E2 -15600.173} C_VEL
LIN {X 0,Y 313.134,Z 167.068,A -85,B 0,C 180,E1 -15603.278,E2 -15603.278} C_VEL
LIN {X 0,Y 312.526,Z 164.56,A -85,B 0,C 180,E1 -15604.208,E2 -15604.208} C_VEL
LIN {X 0,Y 312.514,Z 164.558,A -85,B 0,C 180,E1 -15607.387,E2 -15607.387} C_VEL
LIN {X 0,Y 312.441,Z 164.57,A -85,B 0,C 180,E1 -15610.717,E2 -15610.717} C_VEL
LIN {X 0,Y 312.451,Z 164.564,A -85,B 0,C 180,E1 -15614.21,E2 -15614.21} C_VEL
LIN {X 0,Y 312.456,Z 164.564,A -85,B 0,C 180,E1 -15617.925,E2 -15617.925} C_VEL
LIN {X 0,Y 312.485,Z 164.56,A -85,B 0,C 180,E1 -15621.923,E2 -15621.923} C_VEL
LIN {X 0,Y 312.531,Z 164.55,A -85,B 0,C 180,E1 -15624.22,E2 -15624.22} C_VEL
LIN {X 0,Y 312.503,Z 164.551,A -85,B 0,C 180,E1 -15627.334,E2 -15627.334} C_VEL
LIN {X 0,Y 312.486,Z 164.552,A -85,B 0,C 180,E1 -15631.3,E2 -15631.3} C_VEL
LIN {X 0,Y 312.518,Z 164.546,A -85,B 0,C 180,E1 -15634.705,E2 -15634.705} C_VEL
LIN {X 0,Y 312.541,Z 164.552,A -85,B 0,C 180,E1 -15637.525,E2 -15637.525} C_VEL
LIN {X 0,Y 312.542,Z 164.552,A -85,B 0,C 180,E1 -15641.651,E2 -15641.651} C_VEL
LIN {X 0,Y 312.64,Z 164.537,A -85,B 0,C 180,E1 -15645.684,E2 -15645.684} C_VEL
LIN {X 0,Y 312.684,Z 164.525,A -85,B 0,C 180,E1 -15649.641,E2 -15649.641} C_VEL
LIN {X 0,Y 312.829,Z 164.511,A -85,B 0,C 180,E1 -15652.253,E2 -15652.253} C_VEL
LIN {X 0,Y 312.688,Z 164.532,A -85,B 0,C 180,E1 -15654.842,E2 -15654.842} C_VEL
LIN {X 0,Y 312.969,Z 164.493,A -85,B 0,C 180,E1 -15658.713,E2 -15658.713} C_VEL
LIN {X 0,Y 312.969,Z 164.494,A -85,B 0,C 180,E1 -15661.287,E2 -15661.287} C_VEL
LIN {X 0,Y 312.688,Z 164.531,A -85,B 0,C 180,E1 -15665.158,E2 -15665.158} C_VEL
LIN {X 0,Y 312.799,Z 164.523,A -85,B 0,C 180,E1 -15667.748,E2 -15667.748} C_VEL
LIN {X 0,Y 312.663,Z 164.539,A -85,B 0,C 180,E1 -15671.672,E2 -15671.672} C_VEL
LIN {X 0,Y 312.617,Z 164.543,A -85,B 0,C 180,E1 -15674.828,E2 -15674.828} C_VEL
LIN {X 0,Y 312.536,Z 164.554,A -85,B 0,C 180,E1 -15679.185,E2 -15679.185} C_VEL
LIN {X 0,Y 312.517,Z 164.556,A -85,B 0,C 180,E1 -15682.775,E2 -15682.775} C_VEL
LIN {X 0,Y 312.49,Z 164.565,A -85,B 0,C 180,E1 -15686.731,E2 -15686.731} C_VEL
LIN {X 0,Y 312.536,Z 164.664,A -85,B 0,C 180,E1 -15687.951,E2 -15687.951} C_VEL
LIN {X 0,Y 314.68,Z 173.199,A -85,B 0,C 180,E1 -15690.97,E2 -15690.97} C_VEL
LIN {X 0,Y 322.272,Z 189.992,A -85,B 0,C 180,E1 -15692.243,E2 -15692.243} C_VEL
LIN {X 0,Y 325.489,Z 198.464,A -85,B 0,C 180,E1 -15692.791,E2 -15692.791} C_VEL
LIN {X 0,Y 326.807,Z 205.311,A -85,B 0,C 180,E1 -15693.101,E2 -15693.101} C_VEL
LIN {X 0,Y 324.43,Z 280.901,A -85,B 0,C 180,E1 -15694.904,E2 -15694.904} C_VEL
LIN {X 0,Y 323.561,Z 294.498,A -85,B 0,C 180,E1 -15695.482,E2 -15695.482} C_VEL
LIN {X 0,Y 322.567,Z 306.989,A -85,B 0,C 180,E1 -15696.278,E2 -15696.278} C_VEL
LIN {X 0,Y 321.244,Z 318.605,A -85,B 0,C 180,E1 -15697.269,E2 -15697.269} C_VEL
LIN {X 0,Y 319.727,Z 329.5,A -85,B 0,C 180,E1 -15698.456,E2 -15698.456} C_VEL
LIN {X 0,Y 318.101,Z 340.34,A -85,B 0,C 180,E1 -15699.948,E2 -15699.948} C_VEL
LIN {X 0,Y 316.6,Z 349.341,A -85,B 0,C 180,E1 -15701.5,E2 -15701.5} C_VEL
LIN {X 0,Y 315.102,Z 357.832,A -85,B 0,C 180,E1 -15703.31,E2 -15703.31} C_VEL
LIN {X 0,Y 313.827,Z 364.752,A -85,B 0,C 180,E1 -15705.136,E2 -15705.136} C_VEL
LIN {X 0,Y 312.714,Z 370.892,A -85,B 0,C 180,E1 -15707.168,E2 -15707.168} C_VEL
LIN {X 0,Y 311.883,Z 375.632,A -85,B 0,C 180,E1 -15709.194,E2 -15709.194} C_VEL
LIN {X 0,Y 311.206,Z 379.67,A -85,B 0,C 180,E1 -15711.586,E2 -15711.586} C_VEL
LIN {X 0,Y 310.707,Z 382.261,A -85,B 0,C 180,E1 -15713.977,E2 -15713.977} C_VEL
LIN {X 0,Y 310.487,Z 383.191,A -85,B 0,C 180,E1 -15715.536,E2 -15715.536} C_VEL
LIN {X 0,Y 310.396,Z 383.544,A -85,B 0,C 180,E1 -15717.084,E2 -15717.084} C_VEL
LIN {X 0,Y 310.403,Z 383.043,A -85,B 0,C 180,E1 -15719.36,E2 -15719.36} C_VEL
LIN {X 0,Y 310.645,Z 380.941,A -85,B 0,C 180,E1 -15721.926,E2 -15721.926} C_VEL
LIN {X 0,Y 311.014,Z 378.291,A -85,B 0,C 180,E1 -15723.855,E2 -15723.855} C_VEL
LIN {X 0,Y 311.503,Z 374.066,A -85,B 0,C 180,E1 -15726.039,E2 -15726.039} C_VEL
LIN {X 0,Y 312.089,Z 368.481,A -85,B 0,C 180,E1 -15728.203,E2 -15728.203} C_VEL
LIN {X 0,Y 312.992,Z 361.377,A -85,B 0,C 180,E1 -15730.317,E2 -15730.317} C_VEL
LIN {X 0,Y 314.066,Z 353.951,A -85,B 0,C 180,E1 -15732.08,E2 -15732.08} C_VEL
LIN {X 0,Y 315.335,Z 344.153,A -85,B 0,C 180,E1 -15733.96,E2 -15733.96} C_VEL
LIN {X 0,Y 316.61,Z 333.741,A -85,B 0,C 180,E1 -15735.539,E2 -15735.539} C_VEL
LIN {X 0,Y 317.915,Z 322.491,A -85,B 0,C 180,E1 -15736.897,E2 -15736.897} C_VEL
LIN {X 0,Y 319.027,Z 310.831,A -85,B 0,C 180,E1 -15738,E2 -15738} C_VEL
LIN {X 0,Y 319.922,Z 298.803,A -85,B 0,C 180,E1 -15738.861,E2 -15738.861} C_VEL
LIN {X 0,Y 320.814,Z 285.103,A -85,B 0,C 180,E1 -15739.548,E2 -15739.548} C_VEL
LIN {X 0,Y 321.326,Z 269.824,A -85,B 0,C 180,E1 -15739.995,E2 -15739.995} C_VEL
LIN {X 0,Y 322.854,Z 202.99,A -85,B 0,C 180,E1 -15741.551,E2 -15741.551} C_VEL
LIN {X 0,Y 319.965,Z 188.268,A -85,B 0,C 180,E1 -15742.12,E2 -15742.12} C_VEL
LIN {X 0,Y 314.337,Z 172.393,A -85,B 0,C 180,E1 -15742.936,E2 -15742.936} C_VEL
LIN {X 0,Y 312.698,Z 164.535,A -85,B 0,C 180,E1 -15745.529,E2 -15745.529} C_VEL
LIN {X 0,Y 312.974,Z 164.501,A -85,B 0,C 180,E1 -15748.713,E2 -15748.713} C_VEL
LIN {X 0,Y 312.982,Z 164.496,A -85,B 0,C 180,E1 -15751.287,E2 -15751.287} C_VEL
LIN {X 0,Y 312.844,Z 164.516,A -85,B 0,C 180,E1 -15756.449,E2 -15756.449} C_VEL
LIN {X 0,Y 312.757,Z 164.525,A -85,B 0,C 180,E1 -15759.05,E2 -15759.05} C_VEL
LIN {X 0,Y 312.627,Z 164.54,A -85,B 0,C 180,E1 -15762.991,E2 -15762.991} C_VEL
LIN {X 0,Y 312.581,Z 164.548,A -85,B 0,C 180,E1 -15765.653,E2 -15765.653} C_VEL
LIN {X 0,Y 312.561,Z 164.552,A -85,B 0,C 180,E1 -15769.711,E2 -15769.711} C_VEL
LIN {X 0,Y 312.516,Z 164.552,A -85,B 0,C 180,E1 -15772.775,E2 -15772.775} C_VEL
LIN {X 0,Y 312.488,Z 164.557,A -85,B 0,C 180,E1 -15776.732,E2 -15776.732} C_VEL
LIN {X 0,Y 312.497,Z 164.561,A -85,B 0,C 180,E1 -15779.655,E2 -15779.655} C_VEL
LIN {X 0,Y 312.522,Z 164.553,A -85,B 0,C 180,E1 -15783.689,E2 -15783.689} C_VEL
LIN {X 0,Y 312.516,Z 164.557,A -85,B 0,C 180,E1 -15787.387,E2 -15787.387} C_VEL
LIN {X 0,Y 312.443,Z 164.563,A -85,B 0,C 180,E1 -15790.717,E2 -15790.717} C_VEL
LIN {X 0,Y 312.452,Z 164.558,A -85,B 0,C 180,E1 -15794.21,E2 -15794.21} C_VEL
LIN {X 0,Y 312.462,Z 164.558,A -85,B 0,C 180,E1 -15797.717,E2 -15797.717} C_VEL
LIN {X 0,Y 311.785,Z 164.644,A -85,B 0,C 180,E1 -15798.793,E2 -15798.793} C_VEL
LIN {X 0,Y 308.963,Z 164.998,A -85,B 0,C 180,E1 -15800.546,E2 -15800.546} C_VEL
LIN {X 0,Y 306.578,Z 165.3,A -85,B 0,C 180,E1 -15801.967,E2 -15801.967} C_VEL
LIN {X 0,Y 305.552,Z 165.426,A -85,B 0,C 180,E1 -15803.067,E2 -15803.067} C_VEL
LIN {X 0,Y 305.466,Z 165.434,A -85,B 0,C 180,E1 -15803.44,E2 -15803.44} C_VEL
LIN {X 0,Y 305.467,Z 165.432,A -85,B 0,C 180,E1 -15806.483,E2 -15806.483} C_VEL
LIN {X 0,Y 305.433,Z 165.436,A -85,B 0,C 180,E1 -15809.587,E2 -15809.587} C_VEL
LIN {X 0,Y 305.459,Z 165.436,A -85,B 0,C 180,E1 -15812.602,E2 -15812.602} C_VEL
LIN {X 0,Y 305.476,Z 165.429,A -85,B 0,C 180,E1 -15815.536,E2 -15815.536} C_VEL
LIN {X 0,Y 305.463,Z 165.433,A -85,B 0,C 180,E1 -15818.4,E2 -15818.4} C_VEL
LIN {X 0,Y 305.511,Z 165.427,A -85,B 0,C 180,E1 -15821.213,E2 -15821.213} C_VEL
LIN {X 0,Y 305.582,Z 165.415,A -85,B 0,C 180,E1 -15825.346,E2 -15825.346} C_VEL
LIN {X 0,Y 305.627,Z 165.412,A -85,B 0,C 180,E1 -15829.399,E2 -15829.399} C_VEL
LIN {X 0,Y 305.75,Z 165.399,A -85,B 0,C 180,E1 -15832.073,E2 -15832.073} C_VEL
LIN {X 0,Y 305.661,Z 165.408,A -85,B 0,C 180,E1 -15834.723,E2 -15834.723} C_VEL
LIN {X 0,Y 305.938,Z 165.375,A -85,B 0,C 180,E1 -15838.684,E2 -15838.684} C_VEL
LIN {X 0,Y 305.938,Z 165.372,A -85,B 0,C 180,E1 -15841.316,E2 -15841.316} C_VEL
LIN {X 0,Y 305.79,Z 165.384,A -85,B 0,C 180,E1 -15846.599,E2 -15846.599} C_VEL
LIN {X 0,Y 305.696,Z 165.399,A -85,B 0,C 180,E1 -15849.261,E2 -15849.261} C_VEL
LIN {X 0,Y 305.556,Z 165.422,A -85,B 0,C 180,E1 -15853.297,E2 -15853.297} C_VEL
LIN {X 0,Y 305.495,Z 165.43,A -85,B 0,C 180,E1 -15856.025,E2 -15856.025} C_VEL
LIN {X 0,Y 305.475,Z 165.426,A -85,B 0,C 180,E1 -15860.188,E2 -15860.188} C_VEL
LIN {X 0,Y 305.441,Z 165.435,A -85,B 0,C 180,E1 -15864.467,E2 -15864.467} C_VEL
LIN {X 0,Y 305.442,Z 165.439,A -85,B 0,C 180,E1 -15867.399,E2 -15867.399} C_VEL
LIN {X 0,Y 305.419,Z 165.438,A -85,B 0,C 180,E1 -15870.414,E2 -15870.414} C_VEL
LIN {X 0,Y 305.466,Z 165.432,A -85,B 0,C 180,E1 -15874.078,E2 -15874.078} C_VEL
LIN {X 0,Y 305.455,Z 165.435,A -85,B 0,C 180,E1 -15876.742,E2 -15876.742} C_VEL
LIN {X 0,Y 305.41,Z 165.44,A -85,B 0,C 180,E1 -15880.589,E2 -15880.589} C_VEL
LIN {X 0,Y 305.422,Z 165.439,A -85,B 0,C 180,E1 -15883.656,E2 -15883.656} C_VEL
LIN {X 0,Y 305.435,Z 165.438,A -85,B 0,C 180,E1 -15887.418,E2 -15887.418} C_VEL
LIN {X 0,Y 305.461,Z 165.434,A -85,B 0,C 180,E1 -15891.595,E2 -15891.595} C_VEL
LIN {X 0,Y 305.462,Z 165.437,A -85,B 0,C 180,E1 -15894.886,E2 -15894.886} C_VEL
LIN {X 0,Y 305.459,Z 165.483,A -85,B 0,C 180,E1 -15897.806,E2 -15897.806} C_VEL
LIN {X 0,Y 307.54,Z 175.232,A -85,B 0,C 180,E1 -15900.868,E2 -15900.868} C_VEL
LIN {X 0,Y 309.575,Z 185.936,A -85,B 0,C 180,E1 -15904.086,E2 -15904.086} C_VEL
LIN {X 0,Y 309.671,Z 188.28,A -85,B 0,C 180,E1 -15904.752,E2 -15904.752} C_VEL
LIN {X 0,Y 315.363,Z 225.313,A -85,B 0,C 180,E1 -15906.121,E2 -15906.121} C_VEL
LIN {X 0,Y 315.791,Z 230.03,A -85,B 0,C 180,E1 -15906.27,E2 -15906.27} C_VEL
LIN {X 0,Y 314.042,Z 297.221,A -85,B 0,C 180,E1 -15907.898,E2 -15907.898} C_VEL
LIN {X 0,Y 313.288,Z 310.794,A -85,B 0,C 180,E1 -15908.491,E2 -15908.491} C_VEL
LIN {X 0,Y 312.163,Z 323.627,A -85,B 0,C 180,E1 -15909.317,E2 -15909.317} C_VEL
LIN {X 0,Y 310.862,Z 335.383,A -85,B 0,C 180,E1 -15910.349,E2 -15910.349} C_VEL
LIN {X 0,Y 309.503,Z 346.761,A -85,B 0,C 180,E1 -15911.635,E2 -15911.635} C_VEL
LIN {X 0,Y 308.213,Z 357.077,A -85,B 0,C 180,E1 -15913.107,E2 -15913.107} C_VEL
LIN {X 0,Y 307.047,Z 366.257,A -85,B 0,C 180,E1 -15914.738,E2 -15914.738} C_VEL
LIN {X 0,Y 305.776,Z 375.238,A -85,B 0,C 180,E1 -15916.712,E2 -15916.712} C_VEL
LIN {X 0,Y 304.836,Z 382.44,A -85,B 0,C 180,E1 -15918.699,E2 -15918.699} C_VEL
LIN {X 0,Y 304.228,Z 388.167,A -85,B 0,C 180,E1 -15920.694,E2 -15920.694} C_VEL
LIN {X 0,Y 303.839,Z 392.66,A -85,B 0,C 180,E1 -15922.691,E2 -15922.691} C_VEL
LIN {X 0,Y 303.638,Z 396.048,A -85,B 0,C 180,E1 -15924.688,E2 -15924.688} C_VEL
LIN {X 0,Y 303.63,Z 397.725,A -85,B 0,C 180,E1 -15926.018,E2 -15926.018} C_VEL
LIN {X 0,Y 303.607,Z 398.989,A -85,B 0,C 180,E1 -15927.346,E2 -15927.346} C_VEL
LIN {X 0,Y 303.575,Z 399.841,A -85,B 0,C 180,E1 -15928.673,E2 -15928.673} C_VEL
LIN {X 0,Y 303.604,Z 400.249,A -85,B 0,C 180,E1 -15930,E2 -15930} C_VEL
LIN {X 0,Y 303.601,Z 399.875,A -85,B 0,C 180,E1 -15932.654,E2 -15932.654} C_VEL
LIN {X 0,Y 303.591,Z 399.098,A -85,B 0,C 180,E1 -15933.982,E2 -15933.982} C_VEL
LIN {X 0,Y 303.625,Z 397.613,A -85,B 0,C 180,E1 -15935.545,E2 -15935.545} C_VEL
LIN {X 0,Y 303.99,Z 394.189,A -85,B 0,C 180,E1 -15937.974,E2 -15937.974} C_VEL
LIN {X 0,Y 304.497,Z 390.223,A -85,B 0,C 180,E1 -15939.969,E2 -15939.969} C_VEL
LIN {X 0,Y 305.292,Z 385.128,A -85,B 0,C 180,E1 -15941.958,E2 -15941.958} C_VEL
LIN {X 0,Y 306.508,Z 378.743,A -85,B 0,C 180,E1 -15943.931,E2 -15943.931} C_VEL
LIN {X 0,Y 307.96,Z 370.768,A -85,B 0,C 180,E1 -15945.894,E2 -15945.894} C_VEL
LIN {X 0,Y 309.307,Z 362.668,A -85,B 0,C 180,E1 -15947.522,E2 -15947.522} C_VEL
